LIN {X 0,Y 370.085,Z 646.724,A -85,B 0,C 180,E1 -12842.273,E2 -12842.273} C_VEL
LIN {X 0,Y 368.993,Z 653.125,A -85,B 0,C 180,E1 -12844.625,E2 -12844.625} C_VEL
LIN {X 0,Y 368.227,Z 658.236,A -85,B 0,C 180,E1 -12846.967,E2 -12846.967} C_VEL
LIN {X 0,Y 367.722,Z 662.415,A -85,B 0,C 180,E1 -12849.474,E2 -12849.474} C_VEL
LIN {X 0,Y 367.363,Z 665.468,A -85,B 0,C 180,E1 -12852.176,E2 -12852.176} C_VEL
LIN {X 0,Y 367.23,Z 666.86,A -85,B 0,C 180,E1 -12854.459,E2 -12854.459} C_VEL
LIN {X 0,Y 367.243,Z 667.317,A -85,B 0,C 180,E1 -12856.724,E2 -12856.724} C_VEL
LIN {X 0,Y 367.314,Z 666.714,A -85,B 0,C 180,E1 -12858.969,E2 -12858.969} C_VEL
LIN {X 0,Y 367.306,Z 665.194,A -85,B 0,C 180,E1 -12861.195,E2 -12861.195} C_VEL
LIN {X 0,Y 367.629,Z 662.16,A -85,B 0,C 180,E1 -12863.773,E2 -12863.773} C_VEL
LIN {X 0,Y 368.057,Z 656.967,A -85,B 0,C 180,E1 -12866.716,E2 -12866.716} C_VEL
LIN {X 0,Y 368.653,Z 650.369,A -85,B 0,C 180,E1 -12869.454,E2 -12869.454} C_VEL
LIN {X 0,Y 369.518,Z 643.703,A -85,B 0,C 180,E1 -12871.635,E2 -12871.635} C_VEL
LIN {X 0,Y 370.589,Z 635.761,A -85,B 0,C 180,E1 -12873.806,E2 -12873.806} C_VEL
LIN {X 0,Y 371.387,Z 631.353,A -85,B 0,C 180,E1 -12874.856,E2 -12874.856} C_VEL
LIN {X 0,Y 371.332,Z 628.098,A -85,B 0,C 180,E1 -12875.611,E2 -12875.611} C_VEL
LIN {X 0,Y 367.639,Z 616.959,A -85,B 0,C 180,E1 -12878.099,E2 -12878.099} C_VEL
LIN {X 0,Y 367.616,Z 613.116,A -85,B 0,C 180,E1 -12878.804,E2 -12878.804} C_VEL
LIN {X 0,Y 369.599,Z 601.168,A -85,B 0,C 180,E1 -12880.684,E2 -12880.684} C_VEL
LIN {X 0,Y 371.698,Z 588.051,A -85,B 0,C 180,E1 -12882.42,E2 -12882.42} C_VEL
LIN {X 0,Y 373.867,Z 573.601,A -85,B 0,C 180,E1 -12884.006,E2 -12884.006} C_VEL
LIN {X 0,Y 375.922,Z 559.065,A -85,B 0,C 180,E1 -12885.312,E2 -12885.312} C_VEL
LIN {X 0,Y 377.536,Z 545.128,A -85,B 0,C 180,E1 -12886.353,E2 -12886.353} C_VEL
LIN {X 0,Y 379.089,Z 530.243,A -85,B 0,C 180,E1 -12887.255,E2 -12887.255} C_VEL
LIN {X 0,Y 380.528,Z 513.702,A -85,B 0,C 180,E1 -12888.02,E2 -12888.02} C_VEL
LIN {X 0,Y 381.547,Z 498.273,A -85,B 0,C 180,E1 -12888.526,E2 -12888.526} C_VEL
LIN {X 0,Y 382.324,Z 475.986,A -85,B 0,C 180,E1 -12889.009,E2 -12889.009} C_VEL
LIN {X 0,Y 386.111,Z 337.639,A -85,B 0,C 180,E1 -12891.633,E2 -12891.633} C_VEL
LIN {X 0,Y 376.859,Z 317.995,A -85,B 0,C 180,E1 -12892.926,E2 -12892.926} C_VEL
LIN {X 0,Y 368.621,Z 302.126,A -85,B 0,C 180,E1 -12894.104,E2 -12894.104} C_VEL
LIN {X 0,Y 363.341,Z 293.257,A -85,B 0,C 180,E1 -12894.862,E2 -12894.862} C_VEL
LIN {X 0,Y 362.026,Z 290.544,A -85,B 0,C 180,E1 -12895.068,E2 -12895.068} C_VEL
LIN {X 0,Y 361.859,Z 289.711,A -85,B 0,C 180,E1 -12895.133,E2 -12895.133} C_VEL
LIN {X 0,Y 361.859,Z 289.723,A -85,B 0,C 180,E1 -12899.073,E2 -12899.073} C_VEL
LIN {X 0,Y 361.849,Z 289.725,A -85,B 0,C 180,E1 -12902.945,E2 -12902.945} C_VEL
LIN {X 0,Y 361.865,Z 289.716,A -85,B 0,C 180,E1 -12905.637,E2 -12905.637} C_VEL
LIN {X 0,Y 361.827,Z 289.722,A -85,B 0,C 180,E1 -12909.017,E2 -12909.017} C_VEL
LIN {X 0,Y 361.831,Z 289.72,A -85,B 0,C 180,E1 -12912.83,E2 -12912.83} C_VEL
LIN {X 0,Y 361.814,Z 289.718,A -85,B 0,C 180,E1 -12915.947,E2 -12915.947} C_VEL
LIN {X 0,Y 361.812,Z 289.728,A -85,B 0,C 180,E1 -12919.249,E2 -12919.249} C_VEL
LIN {X 0,Y 361.862,Z 289.676,A -85,B 0,C 180,E1 -12922.981,E2 -12922.981} C_VEL
LIN {X 0,Y 361.859,Z 289.717,A -85,B 0,C 180,E1 -12926.631,E2 -12926.631} C_VEL
LIN {X 0,Y 361.857,Z 289.715,A -85,B 0,C 180,E1 -12929.67,E2 -12929.67} C_VEL
LIN {X 0,Y 361.857,Z 289.724,A -85,B 0,C 180,E1 -12933.467,E2 -12933.467} C_VEL
LIN {X 0,Y 361.866,Z 289.709,A -85,B 0,C 180,E1 -12937.142,E2 -12937.142} C_VEL
LIN {X 0,Y 361.907,Z 289.711,A -85,B 0,C 180,E1 -12940.723,E2 -12940.723} C_VEL
LIN {X 0,Y 361.944,Z 289.711,A -85,B 0,C 180,E1 -12944.225,E2 -12944.225} C_VEL
LIN {X 0,Y 362,Z 289.699,A -85,B 0,C 180,E1 -12946.527,E2 -12946.527} C_VEL
LIN {X 0,Y 362.029,Z 289.7,A -85,B 0,C 180,E1 -12949.937,E2 -12949.937} C_VEL
LIN {X 0,Y 362.15,Z 289.675,A -85,B 0,C 180,E1 -12953.313,E2 -12953.313} C_VEL
LIN {X 0,Y 362.271,Z 289.67,A -85,B 0,C 180,E1 -12957.776,E2 -12957.776} C_VEL
LIN {X 0,Y 362.425,Z 289.634,A -85,B 0,C 180,E1 -12959.999,E2 -12959.999} C_VEL
LIN {X 0,Y 362.281,Z 289.667,A -85,B 0,C 180,E1 -12962.223,E2 -12962.223} C_VEL
LIN {X 0,Y 362.147,Z 289.665,A -85,B 0,C 180,E1 -12966.686,E2 -12966.686} C_VEL
LIN {X 0,Y 362.056,Z 289.688,A -85,B 0,C 180,E1 -12968.933,E2 -12968.933} C_VEL
LIN {X 0,Y 361.96,Z 289.704,A -85,B 0,C 180,E1 -12972.332,E2 -12972.332} C_VEL
LIN {X 0,Y 361.961,Z 289.71,A -85,B 0,C 180,E1 -12974.62,E2 -12974.62} C_VEL
LIN {X 0,Y 361.91,Z 289.715,A -85,B 0,C 180,E1 -12978.101,E2 -12978.101} C_VEL
LIN {X 0,Y 361.891,Z 289.717,A -85,B 0,C 180,E1 -12981.652,E2 -12981.652} C_VEL
LIN {X 0,Y 361.927,Z 289.714,A -85,B 0,C 180,E1 -12985.289,E2 -12985.289} C_VEL
LIN {X 0,Y 361.907,Z 289.713,A -85,B 0,C 180,E1 -12987.779,E2 -12987.779} C_VEL
LIN {X 0,Y 361.836,Z 289.727,A -85,B 0,C 180,E1 -12991.629,E2 -12991.629} C_VEL
LIN {X 0,Y 361.873,Z 289.716,A -85,B 0,C 180,E1 -12995.345,E2 -12995.345} C_VEL
LIN {X 0,Y 361.87,Z 289.724,A -85,B 0,C 180,E1 -12999.027,E2 -12999.027} C_VEL
LIN {X 0,Y 361.835,Z 289.73,A -85,B 0,C 180,E1 -13002.828,E2 -13002.828} C_VEL
LIN {X 0,Y 361.851,Z 289.726,A -85,B 0,C 180,E1 -13005.941,E2 -13005.941} C_VEL
LIN {X 0,Y 361.872,Z 289.883,A -85,B 0,C 180,E1 -13009.425,E2 -13009.425} C_VEL
LIN {X 0,Y 367.396,Z 306.317,A -85,B 0,C 180,E1 -13012.483,E2 -13012.483} C_VEL
LIN {X 0,Y 377.226,Z 326.254,A -85,B 0,C 180,E1 -13013.91,E2 -13013.91} C_VEL
LIN {X 0,Y 384.815,Z 343.06,A -85,B 0,C 180,E1 -13014.983,E2 -13014.983} C_VEL
LIN {X 0,Y 386.007,Z 350.145,A -85,B 0,C 180,E1 -13015.243,E2 -13015.243} C_VEL
LIN {X 0,Y 381.47,Z 514.209,A -85,B 0,C 180,E1 -13018.381,E2 -13018.381} C_VEL
LIN {X 0,Y 380.276,Z 531.49,A -85,B 0,C 180,E1 -13018.914,E2 -13018.914} C_VEL
LIN {X 0,Y 378.832,Z 547.72,A -85,B 0,C 180,E1 -13019.633,E2 -13019.633} C_VEL
LIN {X 0,Y 377.102,Z 563.635,A -85,B 0,C 180,E1 -13020.558,E2 -13020.558} C_VEL
LIN {X 0,Y 375.227,Z 578.232,A -85,B 0,C 180,E1 -13021.616,E2 -13021.616} C_VEL
LIN {X 0,Y 373.014,Z 593.418,A -85,B 0,C 180,E1 -13022.965,E2 -13022.965} C_VEL
LIN {X 0,Y 371.039,Z 607.253,A -85,B 0,C 180,E1 -13024.474,E2 -13024.474} C_VEL
LIN {X 0,Y 368.941,Z 619.349,A -85,B 0,C 180,E1 -13026.025,E2 -13026.025} C_VEL
LIN {X 0,Y 367.037,Z 630.986,A -85,B 0,C 180,E1 -13027.78,E2 -13027.78} C_VEL
LIN {X 0,Y 365.235,Z 642.007,A -85,B 0,C 180,E1 -13029.735,E2 -13029.735} C_VEL
LIN {X 0,Y 363.626,Z 652.593,A -85,B 0,C 180,E1 -13031.987,E2 -13031.987} C_VEL
LIN {X 0,Y 362.341,Z 661.434,A -85,B 0,C 180,E1 -13034.244,E2 -13034.244} C_VEL
LIN {X 0,Y 361.504,Z 668.814,A -85,B 0,C 180,E1 -13036.509,E2 -13036.509} C_VEL
LIN {X 0,Y 360.867,Z 674.908,A -85,B 0,C 180,E1 -13038.77,E2 -13038.77} C_VEL
LIN {X 0,Y 360.456,Z 680.797,A -85,B 0,C 180,E1 -13041.592,E2 -13041.592} C_VEL
LIN {X 0,Y 360.374,Z 684.478,A -85,B 0,C 180,E1 -13044.038,E2 -13044.038} C_VEL
LIN {X 0,Y 360.28,Z 687.094,A -85,B 0,C 180,E1 -13046.645,E2 -13046.645} C_VEL
LIN {X 0,Y 360.315,Z 688.304,A -85,B 0,C 180,E1 -13048.882,E2 -13048.882} C_VEL
LIN {X 0,Y 360.315,Z 688.465,A -85,B 0,C 180,E1 -13051.118,E2 -13051.118} C_VEL
LIN {X 0,Y 360.274,Z 687.726,A -85,B 0,C 180,E1 -13053.355,E2 -13053.355} C_VEL
LIN {X 0,Y 360.374,Z 685.579,A -85,B 0,C 180,E1 -13055.962,E2 -13055.962} C_VEL
LIN {X 0,Y 360.45,Z 683.261,A -85,B 0,C 180,E1 -13057.845,E2 -13057.845} C_VEL
LIN {X 0,Y 360.666,Z 679.474,A -85,B 0,C 180,E1 -13060.101,E2 -13060.101} C_VEL
LIN {X 0,Y 361.249,Z 674.706,A -85,B 0,C 180,E1 -13062.357,E2 -13062.357} C_VEL
LIN {X 0,Y 362.007,Z 668.696,A -85,B 0,C 180,E1 -13064.619,E2 -13064.619} C_VEL
LIN {X 0,Y 363.453,Z 660.481,A -85,B 0,C 180,E1 -13067.151,E2 -13067.151} C_VEL
LIN {X 0,Y 365.086,Z 651.689,A -85,B 0,C 180,E1 -13069.395,E2 -13069.395} C_VEL
LIN {X 0,Y 367.174,Z 641.258,A -85,B 0,C 180,E1 -13071.621,E2 -13071.621} C_VEL
LIN {X 0,Y 369.626,Z 629.387,A -85,B 0,C 180,E1 -13073.732,E2 -13073.732} C_VEL
LIN {X 0,Y 371.938,Z 617.815,A -85,B 0,C 180,E1 -13075.46,E2 -13075.46} C_VEL
LIN {X 0,Y 374.42,Z 605.077,A -85,B 0,C 180,E1 -13077.077,E2 -13077.077} C_VEL
LIN {X 0,Y 377.087,Z 591.395,A -85,B 0,C 180,E1 -13078.523,E2 -13078.523} C_VEL
LIN {X 0,Y 379.398,Z 578,A -85,B 0,C 180,E1 -13079.704,E2 -13079.704} C_VEL
LIN {X 0,Y 381.636,Z 563.787,A -85,B 0,C 180,E1 -13080.733,E2 -13080.733} C_VEL
LIN {X 0,Y 383.646,Z 548.604,A -85,B 0,C 180,E1 -13081.627,E2 -13081.627} C_VEL
LIN {X 0,Y 385.281,Z 533.349,A -85,B 0,C 180,E1 -13082.323,E2 -13082.323} C_VEL
LIN {X 0,Y 386.645,Z 517.043,A -85,B 0,C 180,E1 -13082.852,E2 -13082.852} C_VEL
LIN {X 0,Y 387.657,Z 494.521,A -85,B 0,C 180,E1 -13083.334,E2 -13083.334} C_VEL
LIN {X 0,Y 392.435,Z 351.432,A -85,B 0,C 180,E1 -13086.098,E2 -13086.098} C_VEL
LIN {X 0,Y 391.864,Z 348.162,A -85,B 0,C 180,E1 -13086.244,E2 -13086.244} C_VEL
LIN {X 0,Y 383.625,Z 331.703,A -85,B 0,C 180,E1 -13087.688,E2 -13087.688} C_VEL
LIN {X 0,Y 374.037,Z 314.955,A -85,B 0,C 180,E1 -13089.44,E2 -13089.44} C_VEL
LIN {X 0,Y 367.91,Z 304.9,A -85,B 0,C 180,E1 -13090.637,E2 -13090.637} C_VEL
LIN {X 0,Y 363.24,Z 293.204,A -85,B 0,C 180,E1 -13093.486,E2 -13093.486} C_VEL
LIN {X 0,Y 362.102,Z 290.962,A -85,B 0,C 180,E1 -13094.1,E2 -13094.1} C_VEL
LIN {X 0,Y 361.829,Z 289.716,A -85,B 0,C 180,E1 -13094.409,E2 -13094.409} C_VEL
LIN {X 0,Y 361.835,Z 289.718,A -85,B 0,C 180,E1 -13097.569,E2 -13097.569} C_VEL
LIN {X 0,Y 361.87,Z 289.72,A -85,B 0,C 180,E1 -13100.974,E2 -13100.974} C_VEL
LIN {X 0,Y 361.874,Z 289.722,A -85,B 0,C 180,E1 -13104.656,E2 -13104.656} C_VEL
LIN {X 0,Y 361.837,Z 289.718,A -85,B 0,C 180,E1 -13108.371,E2 -13108.371} C_VEL
LIN {X 0,Y 361.908,Z 289.691,A -85,B 0,C 180,E1 -13112.222,E2 -13112.222} C_VEL
LIN {X 0,Y 361.928,Z 289.716,A -85,B 0,C 180,E1 -13114.711,E2 -13114.711} C_VEL
LIN {X 0,Y 361.862,Z 289.702,A -85,B 0,C 180,E1 -13118.346,E2 -13118.346} C_VEL
LIN {X 0,Y 361.968,Z 289.689,A -85,B 0,C 180,E1 -13122.062,E2 -13122.062} C_VEL
LIN {X 0,Y 361.999,Z 289.705,A -85,B 0,C 180,E1 -13126.102,E2 -13126.102} C_VEL
LIN {X 0,Y 362.001,Z 289.676,A -85,B 0,C 180,E1 -13129.938,E2 -13129.938} C_VEL
LIN {X 0,Y 362.126,Z 289.686,A -85,B 0,C 180,E1 -13133.314,E2 -13133.314} C_VEL
LIN {X 0,Y 362.274,Z 289.665,A -85,B 0,C 180,E1 -13137.777,E2 -13137.777} C_VEL
LIN {X 0,Y 362.363,Z 289.652,A -85,B 0,C 180,E1 -13140.001,E2 -13140.001} C_VEL
LIN {X 0,Y 362.267,Z 289.642,A -85,B 0,C 180,E1 -13142.224,E2 -13142.224} C_VEL
LIN {X 0,Y 362.126,Z 289.675,A -85,B 0,C 180,E1 -13146.688,E2 -13146.688} C_VEL
LIN {X 0,Y 362.002,Z 289.698,A -85,B 0,C 180,E1 -13150.063,E2 -13150.063} C_VEL
LIN {X 0,Y 361.998,Z 289.68,A -85,B 0,C 180,E1 -13153.897,E2 -13153.897} C_VEL
LIN {X 0,Y 361.907,Z 289.703,A -85,B 0,C 180,E1 -13157.908,E2 -13157.908} C_VEL
LIN {X 0,Y 361.856,Z 289.724,A -85,B 0,C 180,E1 -13161.656,E2 -13161.656} C_VEL
LIN {X 0,Y 361.853,Z 289.717,A -85,B 0,C 180,E1 -13165.296,E2 -13165.296} C_VEL
LIN {X 0,Y 361.858,Z 289.711,A -85,B 0,C 180,E1 -13169.074,E2 -13169.074} C_VEL
LIN {X 0,Y 361.848,Z 289.716,A -85,B 0,C 180,E1 -13172.946,E2 -13172.946} C_VEL
LIN {X 0,Y 361.892,Z 289.833,A -85,B 0,C 180,E1 -13175.384,E2 -13175.384} C_VEL
LIN {X 0,Y 362.168,Z 291.049,A -85,B 0,C 180,E1 -13175.523,E2 -13175.523} C_VEL
LIN {X 0,Y 363.591,Z 293.551,A -85,B 0,C 180,E1 -13175.826,E2 -13175.826} C_VEL
LIN {X 0,Y 365.132,Z 295.168,A -85,B 0,C 180,E1 -13176.12,E2 -13176.12} C_VEL
LIN {X 0,Y 367.269,Z 298.449,A -85,B 0,C 180,E1 -13176.547,E2 -13176.547} C_VEL
LIN {X 0,Y 368.815,Z 300.614,A -85,B 0,C 180,E1 -13176.845,E2 -13176.845} C_VEL
LIN {X 0,Y 375.341,Z 310.469,A -85,B 0,C 180,E1 -13178.079,E2 -13178.079} C_VEL
LIN {X 0,Y 384.501,Z 325.897,A -85,B 0,C 180,E1 -13179.732,E2 -13179.732} C_VEL
LIN {X 0,Y 392.18,Z 340.4,A -85,B 0,C 180,E1 -13181.059,E2 -13181.059} C_VEL
LIN {X 0,Y 392.754,Z 342.072,A -85,B 0,C 180,E1 -13181.168,E2 -13181.168} C_VEL
LIN {X 0,Y 387.371,Z 494.991,A -85,B 0,C 180,E1 -13184.129,E2 -13184.129} C_VEL
LIN {X 0,Y 386.172,Z 511.607,A -85,B 0,C 180,E1 -13184.645,E2 -13184.645} C_VEL
LIN {X 0,Y 384.687,Z 527.207,A -85,B 0,C 180,E1 -13185.332,E2 -13185.332} C_VEL
LIN {X 0,Y 382.808,Z 542.708,A -85,B 0,C 180,E1 -13186.219,E2 -13186.219} C_VEL
LIN {X 0,Y 380.595,Z 558.256,A -85,B 0,C 180,E1 -13187.344,E2 -13187.344} C_VEL
LIN {X 0,Y 378.051,Z 573.475,A -85,B 0,C 180,E1 -13188.704,E2 -13188.704} C_VEL
LIN {X 0,Y 375.458,Z 587.611,A -85,B 0,C 180,E1 -13190.255,E2 -13190.255} C_VEL
LIN {X 0,Y 372.987,Z 599.87,A -85,B 0,C 180,E1 -13191.859,E2 -13191.859} C_VEL
LIN {X 0,Y 370.544,Z 611.483,A -85,B 0,C 180,E1 -13193.65,E2 -13193.65} C_VEL
LIN {X 0,Y 368.1,Z 622.784,A -85,B 0,C 180,E1 -13195.72,E2 -13195.72} C_VEL
LIN {X 0,Y 366.207,Z 631.926,A -85,B 0,C 180,E1 -13197.723,E2 -13197.723} C_VEL
LIN {X 0,Y 364.464,Z 640.359,A -85,B 0,C 180,E1 -13199.91,E2 -13199.91} C_VEL
LIN {X 0,Y 363.019,Z 648.046,A -85,B 0,C 180,E1 -13202.313,E2 -13202.313} C_VEL
LIN {X 0,Y 361.908,Z 654.301,A -85,B 0,C 180,E1 -13204.708,E2 -13204.708} C_VEL
LIN {X 0,Y 361.128,Z 659.165,A -85,B 0,C 180,E1 -13207.094,E2 -13207.094} C_VEL
LIN {X 0,Y 360.662,Z 662.879,A -85,B 0,C 180,E1 -13209.466,E2 -13209.466} C_VEL
LIN {X 0,Y 360.294,Z 665.481,A -85,B 0,C 180,E1 -13211.814,E2 -13211.814} C_VEL
LIN {X 0,Y 360.166,Z 666.985,A -85,B 0,C 180,E1 -13214.146,E2 -13214.146} C_VEL
LIN {X 0,Y 360.141,Z 667.536,A -85,B 0,C 180,E1 -13216.457,E2 -13216.457} C_VEL
LIN {X 0,Y 360.213,Z 667.008,A -85,B 0,C 180,E1 -13218.749,E2 -13218.749} C_VEL
LIN {X 0,Y 360.193,Z 665.597,A -85,B 0,C 180,E1 -13221.02,E2 -13221.02} C_VEL
LIN {X 0,Y 360.548,Z 662.44,A -85,B 0,C 180,E1 -13223.79,E2 -13223.79} C_VEL
LIN {X 0,Y 360.785,Z 658.621,A -85,B 0,C 180,E1 -13226.09,E2 -13226.09} C_VEL
LIN {X 0,Y 361.245,Z 653.894,A -85,B 0,C 180,E1 -13228.328,E2 -13228.328} C_VEL
LIN {X 0,Y 362.035,Z 647.944,A -85,B 0,C 180,E1 -13230.556,E2 -13230.556} C_VEL
LIN {X 0,Y 362.947,Z 640.796,A -85,B 0,C 180,E1 -13232.775,E2 -13232.775} C_VEL
LIN {X 0,Y 364.431,Z 631.914,A -85,B 0,C 180,E1 -13235.058,E2 -13235.058} C_VEL
LIN {X 0,Y 366.144,Z 622.083,A -85,B 0,C 180,E1 -13237.167,E2 -13237.167} C_VEL
LIN {X 0,Y 367.616,Z 613.116,A -85,B 0,C 180,E1 -13238.804,E2 -13238.804} C_VEL
LIN {X 0,Y 367.632,Z 609.268,A -85,B 0,C 180,E1 -13239.492,E2 -13239.492} C_VEL
LIN {X 0,Y 364.64,Z 597.528,A -85,B 0,C 180,E1 -13241.553,E2 -13241.553} C_VEL
LIN {X 0,Y 364.371,Z 593.241,A -85,B 0,C 180,E1 -13242.193,E2 -13242.193} C_VEL
LIN {X 0,Y 364.532,Z 591.722,A -85,B 0,C 180,E1 -13242.394,E2 -13242.394} C_VEL
LIN {X 0,Y 366.676,Z 578.023,A -85,B 0,C 180,E1 -13244.003,E2 -13244.003} C_VEL
LIN {X 0,Y 368.775,Z 564.409,A -85,B 0,C 180,E1 -13245.333,E2 -13245.333} C_VEL
LIN {X 0,Y 370.719,Z 549.691,A -85,B 0,C 180,E1 -13246.521,E2 -13246.521} C_VEL
LIN {X 0,Y 372.287,Z 534.616,A -85,B 0,C 180,E1 -13247.51,E2 -13247.51} C_VEL
LIN {X 0,Y 373.878,Z 518.564,A -85,B 0,C 180,E1 -13248.317,E2 -13248.317} C_VEL
LIN {X 0,Y 374.962,Z 503.284,A -85,B 0,C 180,E1 -13248.899,E2 -13248.899} C_VEL
LIN {X 0,Y 375.802,Z 486.805,A -85,B 0,C 180,E1 -13249.316,E2 -13249.316} C_VEL
LIN {X 0,Y 380.045,Z 340.707,A -85,B 0,C 180,E1 -13252.121,E2 -13252.121} C_VEL
LIN {X 0,Y 379.559,Z 338.843,A -85,B 0,C 180,E1 -13252.207,E2 -13252.207} C_VEL
LIN {X 0,Y 370.999,Z 320.605,A -85,B 0,C 180,E1 -13253.441,E2 -13253.441} C_VEL
LIN {X 0,Y 362.905,Z 305.09,A -85,B 0,C 180,E1 -13254.63,E2 -13254.63} C_VEL
LIN {X 0,Y 356.402,Z 294.254,A -85,B 0,C 180,E1 -13255.597,E2 -13255.597} C_VEL
LIN {X 0,Y 355.008,Z 291.577,A -85,B 0,C 180,E1 -13255.819,E2 -13255.819} C_VEL
LIN {X 0,Y 354.823,Z 290.582,A -85,B 0,C 180,E1 -13255.903,E2 -13255.903} C_VEL
LIN {X 0,Y 354.796,Z 290.602,A -85,B 0,C 180,E1 -13259.684,E2 -13259.684} C_VEL
LIN {X 0,Y 354.81,Z 290.604,A -85,B 0,C 180,E1 -13263.702,E2 -13263.702} C_VEL
LIN {X 0,Y 354.795,Z 290.604,A -85,B 0,C 180,E1 -13266.46,E2 -13266.46} C_VEL
LIN {X 0,Y 354.771,Z 290.602,A -85,B 0,C 180,E1 -13269.412,E2 -13269.412} C_VEL
LIN {X 0,Y 354.783,Z 290.598,A -85,B 0,C 180,E1 -13272.865,E2 -13272.865} C_VEL
LIN {X 0,Y 354.763,Z 290.595,A -85,B 0,C 180,E1 -13276.102,E2 -13276.102} C_VEL
LIN {X 0,Y 354.764,Z 290.606,A -85,B 0,C 180,E1 -13279.175,E2 -13279.175} C_VEL
LIN {X 0,Y 354.8,Z 290.56,A -85,B 0,C 180,E1 -13282.404,E2 -13282.404} C_VEL
LIN {X 0,Y 354.809,Z 290.568,A -85,B 0,C 180,E1 -13284.94,E2 -13284.94} C_VEL
LIN {X 0,Y 354.795,Z 290.601,A -85,B 0,C 180,E1 -13288.405,E2 -13288.405} C_VEL
LIN {X 0,Y 354.798,Z 290.59,A -85,B 0,C 180,E1 -13291.614,E2 -13291.614} C_VEL
LIN {X 0,Y 354.835,Z 290.585,A -85,B 0,C 180,E1 -13295.657,E2 -13295.657} C_VEL
LIN {X 0,Y 354.828,Z 290.598,A -85,B 0,C 180,E1 -13299.113,E2 -13299.113} C_VEL
LIN {X 0,Y 354.881,Z 290.578,A -85,B 0,C 180,E1 -13302.718,E2 -13302.718} C_VEL
LIN {X 0,Y 354.953,Z 290.578,A -85,B 0,C 180,E1 -13306.255,E2 -13306.255} C_VEL
LIN {X 0,Y 354.977,Z 290.574,A -85,B 0,C 180,E1 -13309.735,E2 -13309.735} C_VEL
LIN {X 0,Y 355.113,Z 290.553,A -85,B 0,C 180,E1 -13313.18,E2 -13313.18} C_VEL
LIN {X 0,Y 355.234,Z 290.547,A -85,B 0,C 180,E1 -13317.732,E2 -13317.732} C_VEL
LIN {X 0,Y 355.374,Z 290.512,A -85,B 0,C 180,E1 -13319.999,E2 -13319.999} C_VEL
LIN {X 0,Y 355.244,Z 290.543,A -85,B 0,C 180,E1 -13322.267,E2 -13322.267} C_VEL
LIN {X 0,Y 355.113,Z 290.54,A -85,B 0,C 180,E1 -13326.819,E2 -13326.819} C_VEL
LIN {X 0,Y 355.004,Z 290.568,A -85,B 0,C 180,E1 -13329.112,E2 -13329.112} C_VEL
LIN {X 0,Y 354.921,Z 290.581,A -85,B 0,C 180,E1 -13332.58,E2 -13332.58} C_VEL
LIN {X 0,Y 354.886,Z 290.588,A -85,B 0,C 180,E1 -13336.096,E2 -13336.096} C_VEL
LIN {X 0,Y 354.856,Z 290.596,A -85,B 0,C 180,E1 -13339.675,E2 -13339.675} C_VEL
LIN {X 0,Y 354.832,Z 290.602,A -85,B 0,C 180,E1 -13343.336,E2 -13343.336} C_VEL
LIN {X 0,Y 354.886,Z 290.596,A -85,B 0,C 180,E1 -13346.981,E2 -13346.981} C_VEL
LIN {X 0,Y 354.816,Z 290.601,A -85,B 0,C 180,E1 -13349.681,E2 -13349.681} C_VEL
LIN {X 0,Y 354.804,Z 290.601,A -85,B 0,C 180,E1 -13353.702,E2 -13353.702} C_VEL
LIN {X 0,Y 354.797,Z 290.59,A -85,B 0,C 180,E1 -13356.459,E2 -13356.459} C_VEL
LIN {X 0,Y 354.822,Z 290.598,A -85,B 0,C 180,E1 -13359.423,E2 -13359.423} C_VEL
LIN {X 0,Y 354.786,Z 290.607,A -85,B 0,C 180,E1 -13362.867,E2 -13362.867} C_VEL
LIN {X 0,Y 354.794,Z 290.606,A -85,B 0,C 180,E1 -13366.108,E2 -13366.108} C_VEL
LIN {X 0,Y 354.808,Z 290.75,A -85,B 0,C 180,E1 -13368.754,E2 -13368.754} C_VEL
LIN {X 0,Y 359.949,Z 305.875,A -85,B 0,C 180,E1 -13371.688,E2 -13371.688} C_VEL
LIN {X 0,Y 370.514,Z 327.049,A -85,B 0,C 180,E1 -13373.275,E2 -13373.275} C_VEL
LIN {X 0,Y 379.013,Z 345.632,A -85,B 0,C 180,E1 -13374.508,E2 -13374.508} C_VEL
LIN {X 0,Y 379.921,Z 351.835,A -85,B 0,C 180,E1 -13374.728,E2 -13374.728} C_VEL
LIN {X 0,Y 375.254,Z 513.016,A -85,B 0,C 180,E1 -13377.849,E2 -13377.849} C_VEL
LIN {X 0,Y 374.154,Z 529.424,A -85,B 0,C 180,E1 -13378.347,E2 -13378.347} C_VEL
LIN {X 0,Y 372.761,Z 544.864,A -85,B 0,C 180,E1 -13379.006,E2 -13379.006} C_VEL
LIN {X 0,Y 371.128,Z 560.404,A -85,B 0,C 180,E1 -13379.879,E2 -13379.879} C_VEL
LIN {X 0,Y 369.126,Z 575.609,A -85,B 0,C 180,E1 -13380.955,E2 -13380.955} C_VEL
LIN {X 0,Y 366.897,Z 591.109,A -85,B 0,C 180,E1 -13382.321,E2 -13382.321} C_VEL
LIN {X 0,Y 364.804,Z 604.075,A -85,B 0,C 180,E1 -13383.698,E2 -13383.698} C_VEL
LIN {X 0,Y 362.691,Z 616.641,A -85,B 0,C 180,E1 -13385.272,E2 -13385.272} C_VEL
LIN {X 0,Y 360.684,Z 628.685,A -85,B 0,C 180,E1 -13387.064,E2 -13387.064} C_VEL
LIN {X 0,Y 358.691,Z 639.94,A -85,B 0,C 180,E1 -13389.048,E2 -13389.048} C_VEL
LIN {X 0,Y 357.087,Z 650.106,A -85,B 0,C 180,E1 -13391.174,E2 -13391.174} C_VEL
LIN {X 0,Y 355.697,Z 658.932,A -85,B 0,C 180,E1 -13393.352,E2 -13393.352} C_VEL
LIN {X 0,Y 354.698,Z 666.72,A -85,B 0,C 180,E1 -13395.66,E2 -13395.66} C_VEL
LIN {X 0,Y 353.978,Z 673.096,A -85,B 0,C 180,E1 -13397.967,E2 -13397.967} C_VEL
LIN {X 0,Y 353.486,Z 678.302,A -85,B 0,C 180,E1 -13400.271,E2 -13400.271} C_VEL
LIN {X 0,Y 353.356,Z 681.419,A -85,B 0,C 180,E1 -13401.997,E2 -13401.997} C_VEL
LIN {X 0,Y 353.258,Z 684.674,A -85,B 0,C 180,E1 -13404.291,E2 -13404.291} C_VEL
LIN {X 0,Y 353.201,Z 686.845,A -85,B 0,C 180,E1 -13406.578,E2 -13406.578} C_VEL
LIN {X 0,Y 353.216,Z 688.071,A -85,B 0,C 180,E1 -13408.86,E2 -13408.86} C_VEL
LIN {X 0,Y 353.214,Z 688.265,A -85,B 0,C 180,E1 -13411.14,E2 -13411.14} C_VEL
LIN {X 0,Y 353.194,Z 687.543,A -85,B 0,C 180,E1 -13413.422,E2 -13413.422} C_VEL
LIN {X 0,Y 353.273,Z 685.605,A -85,B 0,C 180,E1 -13415.908,E2 -13415.908} C_VEL
LIN {X 0,Y 353.361,Z 683.132,A -85,B 0,C 180,E1 -13418.003,E2 -13418.003} C_VEL
LIN {X 0,Y 353.754,Z 678.308,A -85,B 0,C 180,E1 -13420.879,E2 -13420.879} C_VEL
LIN {X 0,Y 354.465,Z 673.229,A -85,B 0,C 180,E1 -13423.18,E2 -13423.18} C_VEL
LIN {X 0,Y 355.368,Z 667.045,A -85,B 0,C 180,E1 -13425.485,E2 -13425.485} C_VEL
LIN {X 0,Y 357.041,Z 658.483,A -85,B 0,C 180,E1 -13428.061,E2 -13428.061} C_VEL
LIN {X 0,Y 358.791,Z 649.315,A -85,B 0,C 180,E1 -13430.346,E2 -13430.346} C_VEL
LIN {X 0,Y 361.153,Z 638.455,A -85,B 0,C 180,E1 -13432.602,E2 -13432.602} C_VEL
LIN {X 0,Y 363.594,Z 627.204,A -85,B 0,C 180,E1 -13434.569,E2 -13434.569} C_VEL
LIN {X 0,Y 366.182,Z 615.169,A -85,B 0,C 180,E1 -13436.349,E2 -13436.349} C_VEL
LIN {X 0,Y 368.615,Z 603.11,A -85,B 0,C 180,E1 -13437.847,E2 -13437.847} C_VEL
LIN {X 0,Y 371.353,Z 589.187,A -85,B 0,C 180,E1 -13439.303,E2 -13439.303} C_VEL
LIN {X 0,Y 373.815,Z 575.398,A -85,B 0,C 180,E1 -13440.506,E2 -13440.506} C_VEL
LIN {X 0,Y 376.481,Z 558.69,A -85,B 0,C 180,E1 -13441.67,E2 -13441.67} C_VEL
LIN {X 0,Y 378.565,Z 542.077,A -85,B 0,C 180,E1 -13442.574,E2 -13442.574} C_VEL
LIN {X 0,Y 380.194,Z 527.12,A -85,B 0,C 180,E1 -13443.165,E2 -13443.165} C_VEL
LIN {X 0,Y 381.309,Z 512.461,A -85,B 0,C 180,E1 -13443.598,E2 -13443.598} C_VEL
LIN {X 0,Y 386.963,Z 353.291,A -85,B 0,C 180,E1 -13446.73,E2 -13446.73} C_VEL
LIN {X 0,Y 386.544,Z 351.056,A -85,B 0,C 180,E1 -13446.837,E2 -13446.837} C_VEL
LIN {X 0,Y 379.203,Z 336.245,A -85,B 0,C 180,E1 -13448.168,E2 -13448.168} C_VEL
LIN {X 0,Y 369.989,Z 319.961,A -85,B 0,C 180,E1 -13449.904,E2 -13449.904} C_VEL
LIN {X 0,Y 362.878,Z 308.558,A -85,B 0,C 180,E1 -13451.316,E2 -13451.316} C_VEL
LIN {X 0,Y 360.362,Z 304.462,A -85,B 0,C 180,E1 -13451.873,E2 -13451.873} C_VEL
LIN {X 0,Y 355.877,Z 293.535,A -85,B 0,C 180,E1 -13454.689,E2 -13454.689} C_VEL
LIN {X 0,Y 354.791,Z 290.59,A -85,B 0,C 180,E1 -13455.489,E2 -13455.489} C_VEL
LIN {X 0,Y 354.786,Z 290.589,A -85,B 0,C 180,E1 -13459.18,E2 -13459.18} C_VEL
LIN {X 0,Y 354.807,Z 290.583,A -85,B 0,C 180,E1 -13462.403,E2 -13462.403} C_VEL
LIN {X 0,Y 354.812,Z 290.601,A -85,B 0,C 180,E1 -13464.941,E2 -13464.941} C_VEL
LIN {X 0,Y 354.793,Z 290.595,A -85,B 0,C 180,E1 -13468.406,E2 -13468.406} C_VEL
LIN {X 0,Y 354.846,Z 290.57,A -85,B 0,C 180,E1 -13471.619,E2 -13471.619} C_VEL
LIN {X 0,Y 354.899,Z 290.588,A -85,B 0,C 180,E1 -13474.173,E2 -13474.173} C_VEL
LIN {X 0,Y 354.817,Z 290.574,A -85,B 0,C 180,E1 -13477.893,E2 -13477.893} C_VEL
LIN {X 0,Y 354.924,Z 290.569,A -85,B 0,C 180,E1 -13481.892,E2 -13481.892} C_VEL
LIN {X 0,Y 354.944,Z 290.583,A -85,B 0,C 180,E1 -13485.982,E2 -13485.982} C_VEL
LIN {X 0,Y 354.957,Z 290.551,A -85,B 0,C 180,E1 -13489.736,E2 -13489.736} C_VEL
LIN {X 0,Y 355.091,Z 290.563,A -85,B 0,C 180,E1 -13493.18,E2 -13493.18} C_VEL
LIN {X 0,Y 355.236,Z 290.542,A -85,B 0,C 180,E1 -13497.733,E2 -13497.733} C_VEL
LIN {X 0,Y 355.315,Z 290.529,A -85,B 0,C 180,E1 -13500.001,E2 -13500.001} C_VEL
LIN {X 0,Y 355.229,Z 290.518,A -85,B 0,C 180,E1 -13502.268,E2 -13502.268} C_VEL
LIN {X 0,Y 355.091,Z 290.548,A -85,B 0,C 180,E1 -13506.821,E2 -13506.821} C_VEL
LIN {X 0,Y 354.958,Z 290.578,A -85,B 0,C 180,E1 -13510.265,E2 -13510.265} C_VEL
LIN {X 0,Y 354.94,Z 290.558,A -85,B 0,C 180,E1 -13514.016,E2 -13514.016} C_VEL
LIN {X 0,Y 354.847,Z 290.579,A -85,B 0,C 180,E1 -13518.07,E2 -13518.07} C_VEL
LIN {X 0,Y 354.808,Z 290.599,A -85,B 0,C 180,E1 -13522.108,E2 -13522.108} C_VEL
LIN {X 0,Y 354.797,Z 290.602,A -85,B 0,C 180,E1 -13525.836,E2 -13525.836} C_VEL
LIN {X 0,Y 354.795,Z 290.599,A -85,B 0,C 180,E1 -13529.685,E2 -13529.685} C_VEL
LIN {X 0,Y 354.81,Z 290.604,A -85,B 0,C 180,E1 -13533.702,E2 -13533.702} C_VEL
LIN {X 0,Y 354.806,Z 290.602,A -85,B 0,C 180,E1 -13534.241,E2 -13534.241} C_VEL
LIN {X 0,Y 355.81,Z 293.459,A -85,B 0,C 180,E1 -13534.517,E2 -13534.517} C_VEL
LIN {X 0,Y 357.908,Z 295.591,A -85,B 0,C 180,E1 -13534.94,E2 -13534.94} C_VEL
LIN {X 0,Y 360.241,Z 299.311,A -85,B 0,C 180,E1 -13535.439,E2 -13535.439} C_VEL
LIN {X 0,Y 361.6,Z 300.988,A -85,B 0,C 180,E1 -13535.711,E2 -13535.711} C_VEL
LIN {X 0,Y 368.679,Z 311.327,A -85,B 0,C 180,E1 -13537.114,E2 -13537.114} C_VEL
LIN {X 0,Y 377.434,Z 325.766,A -85,B 0,C 180,E1 -13538.77,E2 -13538.77} C_VEL
LIN {X 0,Y 385.685,Z 340.953,A -85,B 0,C 180,E1 -13540.255,E2 -13540.255} C_VEL
LIN {X 0,Y 387.248,Z 344.132,A -85,B 0,C 180,E1 -13540.532,E2 -13540.532} C_VEL
LIN {X 0,Y 381.686,Z 495.648,A -85,B 0,C 180,E1 -13543.504,E2 -13543.504} C_VEL
LIN {X 0,Y 380.49,Z 511.658,A -85,B 0,C 180,E1 -13544.01,E2 -13544.01} C_VEL
LIN {X 0,Y 378.898,Z 527.509,A -85,B 0,C 180,E1 -13544.712,E2 -13544.712} C_VEL
LIN {X 0,Y 376.898,Z 543.343,A -85,B 0,C 180,E1 -13545.632,E2 -13545.632} C_VEL
LIN {X 0,Y 374.601,Z 558.783,A -85,B 0,C 180,E1 -13546.769,E2 -13546.769} C_VEL
LIN {X 0,Y 372.103,Z 573.209,A -85,B 0,C 180,E1 -13548.076,E2 -13548.076} C_VEL
LIN {X 0,Y 369.522,Z 586.482,A -85,B 0,C 180,E1 -13549.533,E2 -13549.533} C_VEL
LIN {X 0,Y 366.72,Z 599.948,A -85,B 0,C 180,E1 -13551.3,E2 -13551.3} C_VEL
LIN {X 0,Y 364.009,Z 612.259,A -85,B 0,C 180,E1 -13553.236,E2 -13553.236} C_VEL
LIN {X 0,Y 361.451,Z 623.491,A -85,B 0,C 180,E1 -13555.345,E2 -13555.345} C_VEL
LIN {X 0,Y 359.256,Z 633.577,A -85,B 0,C 180,E1 -13557.622,E2 -13557.622} C_VEL
LIN {X 0,Y 357.401,Z 641.974,A -85,B 0,C 180,E1 -13559.91,E2 -13559.91} C_VEL
LIN {X 0,Y 355.936,Z 649.254,A -85,B 0,C 180,E1 -13562.314,E2 -13562.314} C_VEL
LIN {X 0,Y 354.794,Z 655.364,A -85,B 0,C 180,E1 -13564.793,E2 -13564.793} C_VEL
LIN {X 0,Y 354.028,Z 660.098,A -85,B 0,C 180,E1 -13567.225,E2 -13567.225} C_VEL
LIN {X 0,Y 353.617,Z 662.893,A -85,B 0,C 180,E1 -13569.086,E2 -13569.086} C_VEL
LIN {X 0,Y 353.246,Z 665.495,A -85,B 0,C 180,E1 -13571.438,E2 -13571.438} C_VEL
LIN {X 0,Y 353.102,Z 667.112,A -85,B 0,C 180,E1 -13573.82,E2 -13573.82} C_VEL
LIN {X 0,Y 353.037,Z 667.719,A -85,B 0,C 180,E1 -13576.179,E2 -13576.179} C_VEL
LIN {X 0,Y 353.11,Z 667.3,A -85,B 0,C 180,E1 -13578.52,E2 -13578.52} C_VEL
LIN {X 0,Y 353.096,Z 665.953,A -85,B 0,C 180,E1 -13580.838,E2 -13580.838} C_VEL
LIN {X 0,Y 353.456,Z 662.695,A -85,B 0,C 180,E1 -13583.824,E2 -13583.824} C_VEL
LIN {X 0,Y 353.677,Z 659.191,A -85,B 0,C 180,E1 -13586.012,E2 -13586.012} C_VEL
LIN {X 0,Y 354.165,Z 654.548,A -85,B 0,C 180,E1 -13588.294,E2 -13588.294} C_VEL
LIN {X 0,Y 355.207,Z 647.098,A -85,B 0,C 180,E1 -13591.134,E2 -13591.134} C_VEL
LIN {X 0,Y 356.359,Z 638.7,A -85,B 0,C 180,E1 -13593.675,E2 -13593.675} C_VEL
LIN {X 0,Y 357.985,Z 629.655,A -85,B 0,C 180,E1 -13595.916,E2 -13595.916} C_VEL
LIN {X 0,Y 359.915,Z 618.94,A -85,B 0,C 180,E1 -13598.139,E2 -13598.139} C_VEL
LIN {X 0,Y 361.792,Z 607.93,A -85,B 0,C 180,E1 -13600.069,E2 -13600.069} C_VEL
LIN {X 0,Y 363.701,Z 596.924,A -85,B 0,C 180,E1 -13601.706,E2 -13601.706} C_VEL
LIN {X 0,Y 364.532,Z 591.722,A -85,B 0,C 180,E1 -13602.394,E2 -13602.394} C_VEL
LIN {X 0,Y 364.628,Z 587.278,A -85,B 0,C 180,E1 -13602.999,E2 -13602.999} C_VEL
LIN {X 0,Y 361.735,Z 572.447,A -85,B 0,C 180,E1 -13605.012,E2 -13605.012} C_VEL
LIN {X 0,Y 361.899,Z 567.484,A -85,B 0,C 180,E1 -13605.536,E2 -13605.536} C_VEL
LIN {X 0,Y 363.832,Z 553.893,A -85,B 0,C 180,E1 -13606.698,E2 -13606.698} C_VEL
LIN {X 0,Y 365.525,Z 539.885,A -85,B 0,C 180,E1 -13607.7,E2 -13607.7} C_VEL
LIN {X 0,Y 367.057,Z 524.632,A -85,B 0,C 180,E1 -13608.561,E2 -13608.561} C_VEL
LIN {X 0,Y 368.393,Z 508.419,A -85,B 0,C 180,E1 -13609.249,E2 -13609.249} C_VEL
LIN {X 0,Y 369.384,Z 491.794,A -85,B 0,C 180,E1 -13609.738,E2 -13609.738} C_VEL
LIN {X 0,Y 373.942,Z 342.873,A -85,B 0,C 180,E1 -13612.651,E2 -13612.651} C_VEL
LIN {X 0,Y 373.518,Z 340.962,A -85,B 0,C 180,E1 -13612.735,E2 -13612.735} C_VEL
LIN {X 0,Y 365.678,Z 324.331,A -85,B 0,C 180,E1 -13613.891,E2 -13613.891} C_VEL
LIN {X 0,Y 358.012,Z 309.528,A -85,B 0,C 180,E1 -13615.05,E2 -13615.05} C_VEL
LIN {X 0,Y 349.318,Z 295.047,A -85,B 0,C 180,E1 -13616.383,E2 -13616.383} C_VEL
LIN {X 0,Y 348.011,Z 292.646,A -85,B 0,C 180,E1 -13616.596,E2 -13616.596} C_VEL
LIN {X 0,Y 347.776,Z 291.463,A -85,B 0,C 180,E1 -13616.68,E2 -13616.68} C_VEL
LIN {X 0,Y 347.732,Z 291.486,A -85,B 0,C 180,E1 -13620.349,E2 -13620.349} C_VEL
LIN {X 0,Y 347.751,Z 291.478,A -85,B 0,C 180,E1 -13624.043,E2 -13624.043} C_VEL
LIN {X 0,Y 347.756,Z 291.478,A -85,B 0,C 180,E1 -13627.321,E2 -13627.321} C_VEL
LIN {X 0,Y 347.698,Z 291.487,A -85,B 0,C 180,E1 -13630.302,E2 -13630.302} C_VEL
LIN {X 0,Y 347.723,Z 291.48,A -85,B 0,C 180,E1 -13633.408,E2 -13633.408} C_VEL
LIN {X 0,Y 347.724,Z 291.47,A -85,B 0,C 180,E1 -13636.686,E2 -13636.686} C_VEL
LIN {X 0,Y 347.702,Z 291.478,A -85,B 0,C 180,E1 -13640.182,E2 -13640.182} C_VEL
LIN {X 0,Y 347.756,Z 291.432,A -85,B 0,C 180,E1 -13642.678,E2 -13642.678} C_VEL
LIN {X 0,Y 347.75,Z 291.461,A -85,B 0,C 180,E1 -13645.956,E2 -13645.956} C_VEL
LIN {X 0,Y 347.74,Z 291.473,A -85,B 0,C 180,E1 -13649.65,E2 -13649.65} C_VEL
LIN {X 0,Y 347.741,Z 291.483,A -85,B 0,C 180,E1 -13653.6,E2 -13653.6} C_VEL
LIN {X 0,Y 347.764,Z 291.463,A -85,B 0,C 180,E1 -13656.159,E2 -13656.159} C_VEL
LIN {X 0,Y 347.808,Z 291.471,A -85,B 0,C 180,E1 -13659.908,E2 -13659.908} C_VEL
LIN {X 0,Y 347.833,Z 291.462,A -85,B 0,C 180,E1 -13663.568,E2 -13663.568} C_VEL
LIN {X 0,Y 347.891,Z 291.452,A -85,B 0,C 180,E1 -13667.16,E2 -13667.16} C_VEL
LIN {X 0,Y 347.941,Z 291.454,A -85,B 0,C 180,E1 -13670.7,E2 -13670.7} C_VEL
LIN {X 0,Y 348.079,Z 291.431,A -85,B 0,C 180,E1 -13673.041,E2 -13673.041} C_VEL
LIN {X 0,Y 348.196,Z 291.424,A -85,B 0,C 180,E1 -13677.686,E2 -13677.686} C_VEL
LIN {X 0,Y 348.324,Z 291.39,A -85,B 0,C 180,E1 -13679.999,E2 -13679.999} C_VEL
LIN {X 0,Y 348.206,Z 291.42,A -85,B 0,C 180,E1 -13682.313,E2 -13682.313} C_VEL
LIN {X 0,Y 348.081,Z 291.414,A -85,B 0,C 180,E1 -13686.958,E2 -13686.958} C_VEL
LIN {X 0,Y 347.945,Z 291.449,A -85,B 0,C 180,E1 -13689.299,E2 -13689.299} C_VEL
LIN {X 0,Y 347.89,Z 291.458,A -85,B 0,C 180,E1 -13692.839,E2 -13692.839} C_VEL
LIN {X 0,Y 347.831,Z 291.467,A -85,B 0,C 180,E1 -13696.431,E2 -13696.431} C_VEL
LIN {X 0,Y 347.811,Z 291.473,A -85,B 0,C 180,E1 -13700.09,E2 -13700.09} C_VEL
LIN {X 0,Y 347.788,Z 291.477,A -85,B 0,C 180,E1 -13703.838,E2 -13703.838} C_VEL
LIN {X 0,Y 347.849,Z 291.469,A -85,B 0,C 180,E1 -13707.254,E2 -13707.254} C_VEL
LIN {X 0,Y 347.747,Z 291.481,A -85,B 0,C 180,E1 -13710.347,E2 -13710.347} C_VEL
LIN {X 0,Y 347.746,Z 291.48,A -85,B 0,C 180,E1 -13714.043,E2 -13714.043} C_VEL
LIN {X 0,Y 347.761,Z 291.468,A -85,B 0,C 180,E1 -13717.32,E2 -13717.32} C_VEL
LIN {X 0,Y 347.73,Z 291.474,A -85,B 0,C 180,E1 -13720.297,E2 -13720.297} C_VEL
LIN {X 0,Y 347.722,Z 291.482,A -85,B 0,C 180,E1 -13723.408,E2 -13723.408} C_VEL
LIN {X 0,Y 347.744,Z 291.477,A -85,B 0,C 180,E1 -13726.682,E2 -13726.682} C_VEL
LIN {X 0,Y 347.755,Z 291.513,A -85,B 0,C 180,E1 -13728.038,E2 -13728.038} C_VEL
LIN {X 0,Y 352.645,Z 305.772,A -85,B 0,C 180,E1 -13730.879,E2 -13730.879} C_VEL
LIN {X 0,Y 363.502,Z 327.169,A -85,B 0,C 180,E1 -13732.566,E2 -13732.566} C_VEL
LIN {X 0,Y 373.216,Z 348.421,A -85,B 0,C 180,E1 -13734.022,E2 -13734.022} C_VEL
LIN {X 0,Y 373.835,Z 353.289,A -85,B 0,C 180,E1 -13734.19,E2 -13734.19} C_VEL
LIN {X 0,Y 369.029,Z 512.983,A -85,B 0,C 180,E1 -13737.326,E2 -13737.326} C_VEL
LIN {X 0,Y 367.888,Z 529.198,A -85,B 0,C 180,E1 -13737.825,E2 -13737.825} C_VEL
LIN {X 0,Y 366.328,Z 545.965,A -85,B 0,C 180,E1 -13738.561,E2 -13738.561} C_VEL
LIN {X 0,Y 364.5,Z 562.203,A -85,B 0,C 180,E1 -13739.514,E2 -13739.514} C_VEL
LIN {X 0,Y 362.581,Z 576.271,A -85,B 0,C 180,E1 -13740.538,E2 -13740.538} C_VEL
LIN {X 0,Y 360.273,Z 591.705,A -85,B 0,C 180,E1 -13741.935,E2 -13741.935} C_VEL
LIN {X 0,Y 357.939,Z 605.657,A -85,B 0,C 180,E1 -13743.469,E2 -13743.469} C_VEL
LIN {X 0,Y 355.626,Z 618.616,A -85,B 0,C 180,E1 -13745.169,E2 -13745.169} C_VEL
LIN {X 0,Y 353.715,Z 629.782,A -85,B 0,C 180,E1 -13746.895,E2 -13746.895} C_VEL
LIN {X 0,Y 351.672,Z 640.884,A -85,B 0,C 180,E1 -13748.917,E2 -13748.917} C_VEL
LIN {X 0,Y 349.894,Z 651.594,A -85,B 0,C 180,E1 -13751.254,E2 -13751.254} C_VEL
LIN {X 0,Y 348.471,Z 660.543,A -85,B 0,C 180,E1 -13753.599,E2 -13753.599} C_VEL
LIN {X 0,Y 347.427,Z 668.595,A -85,B 0,C 180,E1 -13756.16,E2 -13756.16} C_VEL
LIN {X 0,Y 346.801,Z 674.171,A -85,B 0,C 180,E1 -13758.308,E2 -13758.308} C_VEL
LIN {X 0,Y 346.355,Z 679.057,A -85,B 0,C 180,E1 -13760.658,E2 -13760.658} C_VEL
LIN {X 0,Y 346.212,Z 682.906,A -85,B 0,C 180,E1 -13763.004,E2 -13763.004} C_VEL
LIN {X 0,Y 346.138,Z 685.602,A -85,B 0,C 180,E1 -13765.342,E2 -13765.342} C_VEL
LIN {X 0,Y 346.083,Z 687.357,A -85,B 0,C 180,E1 -13767.672,E2 -13767.672} C_VEL
LIN {X 0,Y 346.162,Z 688.06,A -85,B 0,C 180,E1 -13770,E2 -13770} C_VEL
LIN {X 0,Y 346.077,Z 687.858,A -85,B 0,C 180,E1 -13772.328,E2 -13772.328} C_VEL
LIN {X 0,Y 346.118,Z 686.618,A -85,B 0,C 180,E1 -13774.659,E2 -13774.659} C_VEL
LIN {X 0,Y 346.212,Z 684.48,A -85,B 0,C 180,E1 -13776.996,E2 -13776.996} C_VEL
LIN {X 0,Y 346.393,Z 681.267,A -85,B 0,C 180,E1 -13779.341,E2 -13779.341} C_VEL
LIN {X 0,Y 346.883,Z 677.08,A -85,B 0,C 180,E1 -13781.689,E2 -13781.689} C_VEL
LIN {X 0,Y 347.642,Z 671.75,A -85,B 0,C 180,E1 -13784.04,E2 -13784.04} C_VEL
LIN {X 0,Y 348.779,Z 665.253,A -85,B 0,C 180,E1 -13786.386,E2 -13786.386} C_VEL
LIN {X 0,Y 350.404,Z 657.497,A -85,B 0,C 180,E1 -13788.718,E2 -13788.718} C_VEL
LIN {X 0,Y 352.317,Z 648.177,A -85,B 0,C 180,E1 -13791.043,E2 -13791.043} C_VEL
LIN {X 0,Y 354.549,Z 638.609,A -85,B 0,C 180,E1 -13793.048,E2 -13793.048} C_VEL
LIN {X 0,Y 356.991,Z 628.014,A -85,B 0,C 180,E1 -13794.953,E2 -13794.953} C_VEL
LIN {X 0,Y 359.579,Z 616.43,A -85,B 0,C 180,E1 -13796.714,E2 -13796.714} C_VEL
LIN {X 0,Y 362.104,Z 604.677,A -85,B 0,C 180,E1 -13798.235,E2 -13798.235} C_VEL
LIN {X 0,Y 364.87,Z 591.5,A -85,B 0,C 180,E1 -13799.676,E2 -13799.676} C_VEL
LIN {X 0,Y 367.758,Z 576.077,A -85,B 0,C 180,E1 -13801.063,E2 -13801.063} C_VEL
LIN {X 0,Y 370.19,Z 561.512,A -85,B 0,C 180,E1 -13802.112,E2 -13802.112} C_VEL
LIN {X 0,Y 372.367,Z 545.779,A -85,B 0,C 180,E1 -13803.024,E2 -13803.024} C_VEL
LIN {X 0,Y 374.113,Z 530.637,A -85,B 0,C 180,E1 -13803.695,E2 -13803.695} C_VEL
LIN {X 0,Y 375.57,Z 513.757,A -85,B 0,C 180,E1 -13804.224,E2 -13804.224} C_VEL
LIN {X 0,Y 378.377,Z 439.185,A -85,B 0,C 180,E1 -13805.727,E2 -13805.727} C_VEL
LIN {X 0,Y 381.509,Z 354.384,A -85,B 0,C 180,E1 -13807.406,E2 -13807.406} C_VEL
LIN {X 0,Y 374.129,Z 339.5,A -85,B 0,C 180,E1 -13808.789,E2 -13808.789} C_VEL
LIN {X 0,Y 365.406,Z 324.093,A -85,B 0,C 180,E1 -13810.489,E2 -13810.489} C_VEL
LIN {X 0,Y 358.761,Z 313.268,A -85,B 0,C 180,E1 -13811.856,E2 -13811.856} C_VEL
LIN {X 0,Y 352.903,Z 304.066,A -85,B 0,C 180,E1 -13813.169,E2 -13813.169} C_VEL
LIN {X 0,Y 349.181,Z 295.028,A -85,B 0,C 180,E1 -13815.621,E2 -13815.621} C_VEL
LIN {X 0,Y 348.091,Z 292.98,A -85,B 0,C 180,E1 -13816.251,E2 -13816.251} C_VEL
LIN {X 0,Y 347.724,Z 291.484,A -85,B 0,C 180,E1 -13816.687,E2 -13816.687} C_VEL
LIN {X 0,Y 347.746,Z 291.479,A -85,B 0,C 180,E1 -13820.174,E2 -13820.174} C_VEL
LIN {X 0,Y 347.761,Z 291.46,A -85,B 0,C 180,E1 -13822.68,E2 -13822.68} C_VEL
LIN {X 0,Y 347.748,Z 291.466,A -85,B 0,C 180,E1 -13825.957,E2 -13825.957} C_VEL
LIN {X 0,Y 347.749,Z 291.48,A -85,B 0,C 180,E1 -13829.653,E2 -13829.653} C_VEL
LIN {X 0,Y 347.831,Z 291.462,A -85,B 0,C 180,E1 -13833.608,E2 -13833.608} C_VEL
LIN {X 0,Y 347.786,Z 291.456,A -85,B 0,C 180,E1 -13836.162,E2 -13836.162} C_VEL
LIN {X 0,Y 347.812,Z 291.472,A -85,B 0,C 180,E1 -13839.91,E2 -13839.91} C_VEL
LIN {X 0,Y 347.867,Z 291.44,A -85,B 0,C 180,E1 -13842.36,E2 -13842.36} C_VEL
LIN {X 0,Y 347.899,Z 291.461,A -85,B 0,C 180,E1 -13845.971,E2 -13845.971} C_VEL
LIN {X 0,Y 347.897,Z 291.429,A -85,B 0,C 180,E1 -13849.525,E2 -13849.525} C_VEL
LIN {X 0,Y 348.058,Z 291.44,A -85,B 0,C 180,E1 -13853.042,E2 -13853.042} C_VEL
LIN {X 0,Y 348.198,Z 291.417,A -85,B 0,C 180,E1 -13857.687,E2 -13857.687} C_VEL
LIN {X 0,Y 348.267,Z 291.406,A -85,B 0,C 180,E1 -13860.001,E2 -13860.001} C_VEL
LIN {X 0,Y 348.191,Z 291.394,A -85,B 0,C 180,E1 -13862.314,E2 -13862.314} C_VEL
LIN {X 0,Y 348.057,Z 291.421,A -85,B 0,C 180,E1 -13866.959,E2 -13866.959} C_VEL
LIN {X 0,Y 347.899,Z 291.46,A -85,B 0,C 180,E1 -13870.476,E2 -13870.476} C_VEL
LIN {X 0,Y 347.902,Z 291.435,A -85,B 0,C 180,E1 -13874.15,E2 -13874.15} C_VEL
LIN {X 0,Y 347.798,Z 291.454,A -85,B 0,C 180,E1 -13878.243,E2 -13878.243} C_VEL
LIN {X 0,Y 347.766,Z 291.479,A -85,B 0,C 180,E1 -13881.625,E2 -13881.625} C_VEL
LIN {X 0,Y 347.735,Z 291.47,A -85,B 0,C 180,E1 -13885.115,E2 -13885.115} C_VEL
LIN {X 0,Y 347.726,Z 291.467,A -85,B 0,C 180,E1 -13887.702,E2 -13887.702} C_VEL
LIN {X 0,Y 347.732,Z 291.485,A -85,B 0,C 180,E1 -13890.35,E2 -13890.35} C_VEL
LIN {X 0,Y 347.739,Z 291.493,A -85,B 0,C 180,E1 -13892.993,E2 -13892.993} C_VEL
LIN {X 0,Y 348.656,Z 294.183,A -85,B 0,C 180,E1 -13893.248,E2 -13893.248} C_VEL
LIN {X 0,Y 350.703,Z 296.365,A -85,B 0,C 180,E1 -13893.692,E2 -13893.692} C_VEL
LIN {X 0,Y 353.575,Z 300.559,A -85,B 0,C 180,E1 -13894.334,E2 -13894.334} C_VEL
LIN {X 0,Y 354.776,Z 302.032,A -85,B 0,C 180,E1 -13894.589,E2 -13894.589} C_VEL
LIN {X 0,Y 363.907,Z 315.017,A -85,B 0,C 180,E1 -13896.475,E2 -13896.475} C_VEL
LIN {X 0,Y 373.612,Z 331.305,A -85,B 0,C 180,E1 -13898.373,E2 -13898.373} C_VEL
LIN {X 0,Y 381.766,Z 346.552,A -85,B 0,C 180,E1 -13899.881,E2 -13899.881} C_VEL
LIN {X 0,Y 376.12,Z 494.76,A -85,B 0,C 180,E1 -13902.823,E2 -13902.823} C_VEL
LIN {X 0,Y 374.946,Z 510.748,A -85,B 0,C 180,E1 -13903.323,E2 -13903.323} C_VEL
LIN {X 0,Y 373.365,Z 526.083,A -85,B 0,C 180,E1 -13903.985,E2 -13903.985} C_VEL
LIN {X 0,Y 371.37,Z 541.883,A -85,B 0,C 180,E1 -13904.888,E2 -13904.888} C_VEL
LIN {X 0,Y 369.069,Z 556.804,A -85,B 0,C 180,E1 -13905.969,E2 -13905.969} C_VEL
LIN {X 0,Y 366.462,Z 571.448,A -85,B 0,C 180,E1 -13907.279,E2 -13907.279} C_VEL
LIN {X 0,Y 363.737,Z 585.058,A -85,B 0,C 180,E1 -13908.749,E2 -13908.749} C_VEL
LIN {X 0,Y 361.024,Z 597.767,A -85,B 0,C 180,E1 -13910.391,E2 -13910.391} C_VEL
LIN {X 0,Y 358.313,Z 609.714,A -85,B 0,C 180,E1 -13912.226,E2 -13912.226} C_VEL
LIN {X 0,Y 355.65,Z 620.644,A -85,B 0,C 180,E1 -13914.225,E2 -13914.225} C_VEL
LIN {X 0,Y 353.16,Z 631.195,A -85,B 0,C 180,E1 -13916.534,E2 -13916.534} C_VEL
LIN {X 0,Y 351.311,Z 639.349,A -85,B 0,C 180,E1 -13918.659,E2 -13918.659} C_VEL
LIN {X 0,Y 349.525,Z 647.306,A -85,B 0,C 180,E1 -13921.146,E2 -13921.146} C_VEL
LIN {X 0,Y 348.211,Z 653.714,A -85,B 0,C 180,E1 -13923.639,E2 -13923.639} C_VEL
LIN {X 0,Y 347.233,Z 658.83,A -85,B 0,C 180,E1 -13926.121,E2 -13926.121} C_VEL
LIN {X 0,Y 346.587,Z 663.126,A -85,B 0,C 180,E1 -13928.874,E2 -13928.874} C_VEL
LIN {X 0,Y 346.204,Z 665.509,A -85,B 0,C 180,E1 -13931.046,E2 -13931.046} C_VEL
LIN {X 0,Y 346.016,Z 667.241,A -85,B 0,C 180,E1 -13933.479,E2 -13933.479} C_VEL
LIN {X 0,Y 345.947,Z 667.902,A -85,B 0,C 180,E1 -13935.89,E2 -13935.89} C_VEL
LIN {X 0,Y 346.01,Z 667.593,A -85,B 0,C 180,E1 -13938.281,E2 -13938.281} C_VEL
LIN {X 0,Y 345.993,Z 666.297,A -85,B 0,C 180,E1 -13940.648,E2 -13940.648} C_VEL
LIN {X 0,Y 346.241,Z 664.011,A -85,B 0,C 180,E1 -13943.005,E2 -13943.005} C_VEL
LIN {X 0,Y 346.513,Z 660.744,A -85,B 0,C 180,E1 -13945.346,E2 -13945.346} C_VEL
LIN {X 0,Y 346.964,Z 656.401,A -85,B 0,C 180,E1 -13947.678,E2 -13947.678} C_VEL
LIN {X 0,Y 347.582,Z 651.035,A -85,B 0,C 180,E1 -13950,E2 -13950} C_VEL
LIN {X 0,Y 348.577,Z 644.372,A -85,B 0,C 180,E1 -13952.311,E2 -13952.311} C_VEL
LIN {X 0,Y 349.856,Z 636.426,A -85,B 0,C 180,E1 -13954.609,E2 -13954.609} C_VEL
LIN {X 0,Y 351.638,Z 626.965,A -85,B 0,C 180,E1 -13956.887,E2 -13956.887} C_VEL
LIN {X 0,Y 353.478,Z 617.204,A -85,B 0,C 180,E1 -13958.864,E2 -13958.864} C_VEL
LIN {X 0,Y 355.517,Z 605.791,A -85,B 0,C 180,E1 -13960.824,E2 -13960.824} C_VEL
LIN {X 0,Y 357.658,Z 593.385,A -85,B 0,C 180,E1 -13962.627,E2 -13962.627} C_VEL
LIN {X 0,Y 359.889,Z 579.9,A -85,B 0,C 180,E1 -13964.273,E2 -13964.273} C_VEL
LIN {X 0,Y 361.899,Z 567.484,A -85,B 0,C 180,E1 -13965.536,E2 -13965.536} C_VEL
LIN {X 0,Y 362.027,Z 562.511,A -85,B 0,C 180,E1 -13966.043,E2 -13966.043} C_VEL
LIN {X 0,Y 359.237,Z 547.823,A -85,B 0,C 180,E1 -13967.599,E2 -13967.599} C_VEL
LIN {X 0,Y 358.963,Z 542.613,A -85,B 0,C 180,E1 -13968.038,E2 -13968.038} C_VEL
LIN {X 0,Y 359.136,Z 540.823,A -85,B 0,C 180,E1 -13968.165,E2 -13968.165} C_VEL
LIN {X 0,Y 360.722,Z 525.57,A -85,B 0,C 180,E1 -13969.047,E2 -13969.047} C_VEL
LIN {X 0,Y 362.093,Z 509.644,A -85,B 0,C 180,E1 -13969.746,E2 -13969.746} C_VEL
LIN {X 0,Y 363.131,Z 493.631,A -85,B 0,C 180,E1 -13970.24,E2 -13970.24} C_VEL
LIN {X 0,Y 367.932,Z 344.204,A -85,B 0,C 180,E1 -13973.207,E2 -13973.207} C_VEL
LIN {X 0,Y 360.412,Z 328.172,A -85,B 0,C 180,E1 -13974.349,E2 -13974.349} C_VEL
LIN {X 0,Y 353.199,Z 314.044,A -85,B 0,C 180,E1 -13975.473,E2 -13975.473} C_VEL
LIN {X 0,Y 342.412,Z 296.133,A -85,B 0,C 180,E1 -13977.179,E2 -13977.179} C_VEL
LIN {X 0,Y 340.944,Z 293.511,A -85,B 0,C 180,E1 -13977.427,E2 -13977.427} C_VEL
LIN {X 0,Y 340.692,Z 292.357,A -85,B 0,C 180,E1 -13977.496,E2 -13977.496} C_VEL
LIN {X 0,Y 340.685,Z 292.364,A -85,B 0,C 180,E1 -13981.046,E2 -13981.046} C_VEL
LIN {X 0,Y 340.718,Z 292.348,A -85,B 0,C 180,E1 -13985.279,E2 -13985.279} C_VEL
LIN {X 0,Y 340.695,Z 292.351,A -85,B 0,C 180,E1 -13988.382,E2 -13988.382} C_VEL
LIN {X 0,Y 340.692,Z 292.349,A -85,B 0,C 180,E1 -13992.043,E2 -13992.043} C_VEL
LIN {X 0,Y 340.651,Z 292.351,A -85,B 0,C 180,E1 -13996.227,E2 -13996.227} C_VEL
LIN {X 0,Y 340.67,Z 292.362,A -85,B 0,C 180,E1 -13998.687,E2 -13998.687} C_VEL
LIN {X 0,Y 340.72,Z 292.321,A -85,B 0,C 180,E1 -14001.77,E2 -14001.77} C_VEL
LIN {X 0,Y 340.724,Z 292.331,A -85,B 0,C 180,E1 -14005.595,E2 -14005.595} C_VEL
LIN {X 0,Y 340.695,Z 292.357,A -85,B 0,C 180,E1 -14008.954,E2 -14008.954} C_VEL
LIN {X 0,Y 340.713,Z 292.354,A -85,B 0,C 180,E1 -14013.011,E2 -14013.011} C_VEL
LIN {X 0,Y 340.74,Z 292.34,A -85,B 0,C 180,E1 -14015.636,E2 -14015.636} C_VEL
LIN {X 0,Y 340.736,Z 292.356,A -85,B 0,C 180,E1 -14019.473,E2 -14019.473} C_VEL
LIN {X 0,Y 340.794,Z 292.33,A -85,B 0,C 180,E1 -14021.98,E2 -14021.98} C_VEL
LIN {X 0,Y 340.871,Z 292.336,A -85,B 0,C 180,E1 -14025.704,E2 -14025.704} C_VEL
LIN {X 0,Y 340.871,Z 292.325,A -85,B 0,C 180,E1 -14029.306,E2 -14029.306} C_VEL
LIN {X 0,Y 341.046,Z 292.309,A -85,B 0,C 180,E1 -14032.897,E2 -14032.897} C_VEL
LIN {X 0,Y 341.157,Z 292.302,A -85,B 0,C 180,E1 -14037.638,E2 -14037.638} C_VEL
LIN {X 0,Y 341.275,Z 292.268,A -85,B 0,C 180,E1 -14039.999,E2 -14039.999} C_VEL
LIN {X 0,Y 341.168,Z 292.297,A -85,B 0,C 180,E1 -14042.361,E2 -14042.361} C_VEL
LIN {X 0,Y 341.051,Z 292.289,A -85,B 0,C 180,E1 -14047.102,E2 -14047.102} C_VEL
LIN {X 0,Y 340.871,Z 292.337,A -85,B 0,C 180,E1 -14050.693,E2 -14050.693} C_VEL
LIN {X 0,Y 340.862,Z 292.338,A -85,B 0,C 180,E1 -14054.324,E2 -14054.324} C_VEL
LIN {X 0,Y 340.785,Z 292.348,A -85,B 0,C 180,E1 -14058.44,E2 -14058.44} C_VEL
LIN {X 0,Y 340.753,Z 292.349,A -85,B 0,C 180,E1 -14061.856,E2 -14061.856} C_VEL
LIN {X 0,Y 340.771,Z 292.35,A -85,B 0,C 180,E1 -14065.664,E2 -14065.664} C_VEL
LIN {X 0,Y 340.727,Z 292.351,A -85,B 0,C 180,E1 -14068.32,E2 -14068.32} C_VEL
LIN {X 0,Y 340.696,Z 292.358,A -85,B 0,C 180,E1 -14071.044,E2 -14071.044} C_VEL
LIN {X 0,Y 340.717,Z 292.352,A -85,B 0,C 180,E1 -14075.278,E2 -14075.278} C_VEL
LIN {X 0,Y 340.708,Z 292.357,A -85,B 0,C 180,E1 -14078.386,E2 -14078.386} C_VEL
LIN {X 0,Y 340.697,Z 292.358,A -85,B 0,C 180,E1 -14082.045,E2 -14082.045} C_VEL
LIN {X 0,Y 340.689,Z 292.359,A -85,B 0,C 180,E1 -14085.462,E2 -14085.462} C_VEL
LIN {X 0,Y 340.73,Z 292.466,A -85,B 0,C 180,E1 -14087.324,E2 -14087.324} C_VEL
LIN {X 0,Y 345.327,Z 305.639,A -85,B 0,C 180,E1 -14090.028,E2 -14090.028} C_VEL
LIN {X 0,Y 356.476,Z 327.312,A -85,B 0,C 180,E1 -14091.826,E2 -14091.826} C_VEL
LIN {X 0,Y 366.771,Z 349.521,A -85,B 0,C 180,E1 -14093.417,E2 -14093.417} C_VEL
LIN {X 0,Y 367.503,Z 351.56,A -85,B 0,C 180,E1 -14093.536,E2 -14093.536} C_VEL
LIN {X 0,Y 367.752,Z 355.324,A -85,B 0,C 180,E1 -14093.647,E2 -14093.647} C_VEL
LIN {X 0,Y 362.791,Z 513.563,A -85,B 0,C 180,E1 -14096.801,E2 -14096.801} C_VEL
LIN {X 0,Y 361.534,Z 530.757,A -85,B 0,C 180,E1 -14097.354,E2 -14097.354} C_VEL
LIN {X 0,Y 359.923,Z 547.026,A -85,B 0,C 180,E1 -14098.1,E2 -14098.1} C_VEL
LIN {X 0,Y 358.037,Z 562.978,A -85,B 0,C 180,E1 -14099.067,E2 -14099.067} C_VEL
LIN {X 0,Y 356.055,Z 576.873,A -85,B 0,C 180,E1 -14100.106,E2 -14100.106} C_VEL
LIN {X 0,Y 353.693,Z 592.131,A -85,B 0,C 180,E1 -14101.518,E2 -14101.518} C_VEL
LIN {X 0,Y 351.26,Z 606.04,A -85,B 0,C 180,E1 -14103.084,E2 -14103.084} C_VEL
LIN {X 0,Y 349.074,Z 617.907,A -85,B 0,C 180,E1 -14104.67,E2 -14104.67} C_VEL
LIN {X 0,Y 347.061,Z 629.154,A -85,B 0,C 180,E1 -14106.426,E2 -14106.426} C_VEL
LIN {X 0,Y 344.918,Z 640.294,A -85,B 0,C 180,E1 -14108.484,E2 -14108.484} C_VEL
LIN {X 0,Y 343.07,Z 651.072,A -85,B 0,C 180,E1 -14110.867,E2 -14110.867} C_VEL
LIN {X 0,Y 341.527,Z 660.083,A -85,B 0,C 180,E1 -14113.256,E2 -14113.256} C_VEL
LIN {X 0,Y 340.504,Z 667.619,A -85,B 0,C 180,E1 -14115.66,E2 -14115.66} C_VEL
LIN {X 0,Y 339.776,Z 673.797,A -85,B 0,C 180,E1 -14118.063,E2 -14118.063} C_VEL
LIN {X 0,Y 339.283,Z 678.724,A -85,B 0,C 180,E1 -14120.461,E2 -14120.461} C_VEL
LIN {X 0,Y 339.125,Z 682.608,A -85,B 0,C 180,E1 -14122.857,E2 -14122.857} C_VEL
LIN {X 0,Y 339.041,Z 685.329,A -85,B 0,C 180,E1 -14125.244,E2 -14125.244} C_VEL
LIN {X 0,Y 338.997,Z 687.122,A -85,B 0,C 180,E1 -14127.624,E2 -14127.624} C_VEL
LIN {X 0,Y 339.065,Z 687.843,A -85,B 0,C 180,E1 -14130,E2 -14130} C_VEL
LIN {X 0,Y 338.991,Z 687.676,A -85,B 0,C 180,E1 -14132.377,E2 -14132.377} C_VEL
LIN {X 0,Y 339.021,Z 686.454,A -85,B 0,C 180,E1 -14134.757,E2 -14134.757} C_VEL
LIN {X 0,Y 339.126,Z 684.352,A -85,B 0,C 180,E1 -14137.143,E2 -14137.143} C_VEL
LIN {X 0,Y 339.321,Z 681.162,A -85,B 0,C 180,E1 -14139.538,E2 -14139.538} C_VEL
LIN {X 0,Y 339.872,Z 677.021,A -85,B 0,C 180,E1 -14141.934,E2 -14141.934} C_VEL
LIN {X 0,Y 340.66,Z 671.715,A -85,B 0,C 180,E1 -14144.334,E2 -14144.334} C_VEL
LIN {X 0,Y 341.876,Z 665.265,A -85,B 0,C 180,E1 -14146.726,E2 -14146.726} C_VEL
LIN {X 0,Y 343.586,Z 657.547,A -85,B 0,C 180,E1 -14149.104,E2 -14149.104} C_VEL
LIN {X 0,Y 345.628,Z 648.275,A -85,B 0,C 180,E1 -14151.47,E2 -14151.47} C_VEL
LIN {X 0,Y 347.96,Z 638.783,A -85,B 0,C 180,E1 -14153.51,E2 -14153.51} C_VEL
LIN {X 0,Y 350.71,Z 627.285,A -85,B 0,C 180,E1 -14155.609,E2 -14155.609} C_VEL
LIN {X 0,Y 353.691,Z 614.795,A -85,B 0,C 180,E1 -14157.516,E2 -14157.516} C_VEL
LIN {X 0,Y 356.155,Z 603.919,A -85,B 0,C 180,E1 -14158.912,E2 -14158.912} C_VEL
LIN {X 0,Y 359.064,Z 590.263,A -85,B 0,C 180,E1 -14160.41,E2 -14160.41} C_VEL
LIN {X 0,Y 362.024,Z 575.088,A -85,B 0,C 180,E1 -14161.775,E2 -14161.775} C_VEL
LIN {X 0,Y 364.877,Z 558.426,A -85,B 0,C 180,E1 -14162.965,E2 -14162.965} C_VEL
LIN {X 0,Y 367.146,Z 541.861,A -85,B 0,C 180,E1 -14163.885,E2 -14163.885} C_VEL
LIN {X 0,Y 369.027,Z 525.217,A -85,B 0,C 180,E1 -14164.554,E2 -14164.554} C_VEL
LIN {X 0,Y 370.279,Z 508.693,A -85,B 0,C 180,E1 -14165.015,E2 -14165.015} C_VEL
LIN {X 0,Y 376.143,Z 356.929,A -85,B 0,C 180,E1 -14168.062,E2 -14168.062} C_VEL
LIN {X 0,Y 369.135,Z 342.856,A -85,B 0,C 180,E1 -14169.421,E2 -14169.421} C_VEL
LIN {X 0,Y 361.039,Z 328.486,A -85,B 0,C 180,E1 -14171.054,E2 -14171.054} C_VEL
LIN {X 0,Y 354.91,Z 318.382,A -85,B 0,C 180,E1 -14172.356,E2 -14172.356} C_VEL
LIN {X 0,Y 348.142,Z 308.016,A -85,B 0,C 180,E1 -14173.869,E2 -14173.869} C_VEL
LIN {X 0,Y 345.335,Z 303.683,A -85,B 0,C 180,E1 -14174.579,E2 -14174.579} C_VEL
LIN {X 0,Y 342.036,Z 295.718,A -85,B 0,C 180,E1 -14176.872,E2 -14176.872} C_VEL
LIN {X 0,Y 340.898,Z 293.382,A -85,B 0,C 180,E1 -14177.609,E2 -14177.609} C_VEL
LIN {X 0,Y 340.698,Z 292.344,A -85,B 0,C 180,E1 -14177.955,E2 -14177.955} C_VEL
LIN {X 0,Y 340.732,Z 292.339,A -85,B 0,C 180,E1 -14181.773,E2 -14181.773} C_VEL
LIN {X 0,Y 340.722,Z 292.346,A -85,B 0,C 180,E1 -14185.596,E2 -14185.596} C_VEL
LIN {X 0,Y 340.698,Z 292.356,A -85,B 0,C 180,E1 -14188.956,E2 -14188.956} C_VEL
LIN {X 0,Y 340.803,Z 292.325,A -85,B 0,C 180,E1 -14193.021,E2 -14193.021} C_VEL
LIN {X 0,Y 340.755,Z 292.341,A -85,B 0,C 180,E1 -14195.639,E2 -14195.639} C_VEL
LIN {X 0,Y 340.739,Z 292.35,A -85,B 0,C 180,E1 -14199.474,E2 -14199.474} C_VEL
LIN {X 0,Y 340.859,Z 292.317,A -85,B 0,C 180,E1 -14201.985,E2 -14201.985} C_VEL
LIN {X 0,Y 340.87,Z 292.336,A -85,B 0,C 180,E1 -14205.706,E2 -14205.706} C_VEL
LIN {X 0,Y 340.849,Z 292.306,A -85,B 0,C 180,E1 -14209.306,E2 -14209.306} C_VEL
LIN {X 0,Y 341.004,Z 292.319,A -85,B 0,C 180,E1 -14212.897,E2 -14212.897} C_VEL
LIN {X 0,Y 340.828,Z 292.308,A -85,B 0,C 180,E1 -14215.269,E2 -14215.269} C_VEL
LIN {X 0,Y 341.159,Z 292.291,A -85,B 0,C 180,E1 -14217.639,E2 -14217.639} C_VEL
LIN {X 0,Y 341.219,Z 292.283,A -85,B 0,C 180,E1 -14220.001,E2 -14220.001} C_VEL
LIN {X 0,Y 341.128,Z 292.273,A -85,B 0,C 180,E1 -14222.362,E2 -14222.362} C_VEL
LIN {X 0,Y 340.993,Z 292.305,A -85,B 0,C 180,E1 -14226.542,E2 -14226.542} C_VEL
LIN {X 0,Y 340.884,Z 292.318,A -85,B 0,C 180,E1 -14229.494,E2 -14229.494} C_VEL
LIN {X 0,Y 340.846,Z 292.316,A -85,B 0,C 180,E1 -14233.11,E2 -14233.11} C_VEL
LIN {X 0,Y 340.801,Z 292.336,A -85,B 0,C 180,E1 -14235.551,E2 -14235.551} C_VEL
LIN {X 0,Y 340.711,Z 292.331,A -85,B 0,C 180,E1 -14239.272,E2 -14239.272} C_VEL
LIN {X 0,Y 340.702,Z 292.342,A -85,B 0,C 180,E1 -14243.076,E2 -14243.076} C_VEL
LIN {X 0,Y 340.712,Z 292.348,A -85,B 0,C 180,E1 -14246.989,E2 -14246.989} C_VEL
LIN {X 0,Y 340.719,Z 292.356,A -85,B 0,C 180,E1 -14249.964,E2 -14249.964} C_VEL
LIN {X 0,Y 340.719,Z 292.535,A -85,B 0,C 180,E1 -14251.649,E2 -14251.649} C_VEL
LIN {X 0,Y 341.557,Z 294.979,A -85,B 0,C 180,E1 -14251.898,E2 -14251.898} C_VEL
LIN {X 0,Y 343.489,Z 297.128,A -85,B 0,C 180,E1 -14252.352,E2 -14252.352} C_VEL
LIN {X 0,Y 344.3,Z 297.941,A -85,B 0,C 180,E1 -14252.537,E2 -14252.537} C_VEL
LIN {X 0,Y 346.269,Z 301.097,A -85,B 0,C 180,E1 -14253.014,E2 -14253.014} C_VEL
LIN {X 0,Y 347.922,Z 302.977,A -85,B 0,C 180,E1 -14253.382,E2 -14253.382} C_VEL
LIN {X 0,Y 350.508,Z 306.547,A -85,B 0,C 180,E1 -14253.966,E2 -14253.966} C_VEL
LIN {X 0,Y 359.975,Z 320.02,A -85,B 0,C 180,E1 -14255.983,E2 -14255.983} C_VEL
LIN {X 0,Y 369.284,Z 335.883,A -85,B 0,C 180,E1 -14257.863,E2 -14257.863} C_VEL
LIN {X 0,Y 376.378,Z 349.221,A -85,B 0,C 180,E1 -14259.222,E2 -14259.222} C_VEL
LIN {X 0,Y 370.544,Z 495.661,A -85,B 0,C 180,E1 -14262.162,E2 -14262.162} C_VEL
LIN {X 0,Y 369.269,Z 511.884,A -85,B 0,C 180,E1 -14262.683,E2 -14262.683} C_VEL
LIN {X 0,Y 367.538,Z 527.762,A -85,B 0,C 180,E1 -14263.395,E2 -14263.395} C_VEL
LIN {X 0,Y 365.439,Z 543.225,A -85,B 0,C 180,E1 -14264.306,E2 -14264.306} C_VEL
LIN {X 0,Y 363.022,Z 558.314,A -85,B 0,C 180,E1 -14265.429,E2 -14265.429} C_VEL
LIN {X 0,Y 360.275,Z 572.947,A -85,B 0,C 180,E1 -14266.778,E2 -14266.778} C_VEL
LIN {X 0,Y 357.518,Z 586.073,A -85,B 0,C 180,E1 -14268.238,E2 -14268.238} C_VEL
LIN {X 0,Y 354.403,Z 599.72,A -85,B 0,C 180,E1 -14270.058,E2 -14270.058} C_VEL
LIN {X 0,Y 351.425,Z 612.129,A -85,B 0,C 180,E1 -14272.051,E2 -14272.051} C_VEL
LIN {X 0,Y 348.624,Z 623.418,A -85,B 0,C 180,E1 -14274.224,E2 -14274.224} C_VEL
LIN {X 0,Y 346.314,Z 632.497,A -85,B 0,C 180,E1 -14276.31,E2 -14276.31} C_VEL
LIN {X 0,Y 344.258,Z 640.963,A -85,B 0,C 180,E1 -14278.629,E2 -14278.629} C_VEL
LIN {X 0,Y 342.443,Z 648.647,A -85,B 0,C 180,E1 -14281.165,E2 -14281.165} C_VEL
LIN {X 0,Y 341.118,Z 654.905,A -85,B 0,C 180,E1 -14283.707,E2 -14283.707} C_VEL
LIN {X 0,Y 340.135,Z 659.773,A -85,B 0,C 180,E1 -14286.239,E2 -14286.239} C_VEL
LIN {X 0,Y 339.539,Z 663.377,A -85,B 0,C 180,E1 -14288.662,E2 -14288.662} C_VEL
LIN {X 0,Y 339.181,Z 665.527,A -85,B 0,C 180,E1 -14290.638,E2 -14290.638} C_VEL
LIN {X 0,Y 338.96,Z 667.365,A -85,B 0,C 180,E1 -14293.125,E2 -14293.125} C_VEL
LIN {X 0,Y 338.856,Z 668.085,A -85,B 0,C 180,E1 -14295.588,E2 -14295.588} C_VEL
LIN {X 0,Y 338.918,Z 667.885,A -85,B 0,C 180,E1 -14298.032,E2 -14298.032} C_VEL
LIN {X 0,Y 338.885,Z 666.643,A -85,B 0,C 180,E1 -14300.45,E2 -14300.45} C_VEL
LIN {X 0,Y 339.127,Z 664.466,A -85,B 0,C 180,E1 -14302.857,E2 -14302.857} C_VEL
LIN {X 0,Y 339.428,Z 661.251,A -85,B 0,C 180,E1 -14305.249,E2 -14305.249} C_VEL
LIN {X 0,Y 339.875,Z 657.022,A -85,B 0,C 180,E1 -14307.63,E2 -14307.63} C_VEL
LIN {X 0,Y 340.489,Z 651.719,A -85,B 0,C 180,E1 -14310,E2 -14310} C_VEL
LIN {X 0,Y 341.53,Z 645.169,A -85,B 0,C 180,E1 -14312.359,E2 -14312.359} C_VEL
LIN {X 0,Y 342.817,Z 637.361,A -85,B 0,C 180,E1 -14314.704,E2 -14314.704} C_VEL
LIN {X 0,Y 344.649,Z 628.043,A -85,B 0,C 180,E1 -14317.028,E2 -14317.028} C_VEL
LIN {X 0,Y 346.817,Z 616.915,A -85,B 0,C 180,E1 -14319.33,E2 -14319.33} C_VEL
LIN {X 0,Y 348.961,Z 605.401,A -85,B 0,C 180,E1 -14321.324,E2 -14321.324} C_VEL
LIN {X 0,Y 351.223,Z 592.872,A -85,B 0,C 180,E1 -14323.157,E2 -14323.157} C_VEL
LIN {X 0,Y 353.535,Z 579.241,A -85,B 0,C 180,E1 -14324.829,E2 -14324.829} C_VEL
LIN {X 0,Y 355.778,Z 565.78,A -85,B 0,C 180,E1 -14326.202,E2 -14326.202} C_VEL
LIN {X 0,Y 357.859,Z 551.164,A -85,B 0,C 180,E1 -14327.427,E2 -14327.427} C_VEL
LIN {X 0,Y 359.136,Z 540.823,A -85,B 0,C 180,E1 -14328.165,E2 -14328.165} C_VEL
LIN {X 0,Y 359.258,Z 535.454,A -85,B 0,C 180,E1 -14328.559,E2 -14328.559} C_VEL
LIN {X 0,Y 357.628,Z 526.747,A -85,B 0,C 180,E1 -14329.279,E2 -14329.279} C_VEL
LIN {X 0,Y 355.849,Z 517.864,A -85,B 0,C 180,E1 -14329.928,E2 -14329.928} C_VEL
LIN {X 0,Y 355.719,Z 512.222,A -85,B 0,C 180,E1 -14330.208,E2 -14330.208} C_VEL
LIN {X 0,Y 356.904,Z 495.465,A -85,B 0,C 180,E1 -14330.76,E2 -14330.76} C_VEL
LIN {X 0,Y 361.415,Z 359.866,A -85,B 0,C 180,E1 -14333.5,E2 -14333.5} C_VEL
LIN {X 0,Y 361.734,Z 345.882,A -85,B 0,C 180,E1 -14333.794,E2 -14333.794} C_VEL
LIN {X 0,Y 352.839,Z 327.15,A -85,B 0,C 180,E1 -14335.193,E2 -14335.193} C_VEL
LIN {X 0,Y 347.766,Z 317.52,A -85,B 0,C 180,E1 -14336.003,E2 -14336.003} C_VEL
LIN {X 0,Y 337.625,Z 300.653,A -85,B 0,C 180,E1 -14337.656,E2 -14337.656} C_VEL
LIN {X 0,Y 335.629,Z 297.357,A -85,B 0,C 180,E1 -14337.997,E2 -14337.997} C_VEL
LIN {X 0,Y 334.037,Z 294.848,A -85,B 0,C 180,E1 -14338.269,E2 -14338.269} C_VEL
LIN {X 0,Y 333.634,Z 293.245,A -85,B 0,C 180,E1 -14338.376,E2 -14338.376} C_VEL
LIN {X 0,Y 333.623,Z 293.237,A -85,B 0,C 180,E1 -14341.779,E2 -14341.779} C_VEL
LIN {X 0,Y 333.687,Z 293.224,A -85,B 0,C 180,E1 -14344.773,E2 -14344.773} C_VEL
LIN {X 0,Y 333.645,Z 293.231,A -85,B 0,C 180,E1 -14347.652,E2 -14347.652} C_VEL
LIN {X 0,Y 333.605,Z 293.24,A -85,B 0,C 180,E1 -14350.773,E2 -14350.773} C_VEL
LIN {X 0,Y 333.592,Z 293.245,A -85,B 0,C 180,E1 -14354.249,E2 -14354.249} C_VEL
LIN {X 0,Y 333.637,Z 293.23,A -85,B 0,C 180,E1 -14357.617,E2 -14357.617} C_VEL
LIN {X 0,Y 333.617,Z 293.214,A -85,B 0,C 180,E1 -14361.21,E2 -14361.21} C_VEL
LIN {X 0,Y 333.674,Z 293.182,A -85,B 0,C 180,E1 -14363.86,E2 -14363.86} C_VEL
LIN {X 0,Y 333.645,Z 293.233,A -85,B 0,C 180,E1 -14367.412,E2 -14367.412} C_VEL
LIN {X 0,Y 333.633,Z 293.222,A -85,B 0,C 180,E1 -14371.02,E2 -14371.02} C_VEL
LIN {X 0,Y 333.696,Z 293.224,A -85,B 0,C 180,E1 -14375.087,E2 -14375.087} C_VEL
LIN {X 0,Y 333.668,Z 293.233,A -85,B 0,C 180,E1 -14379.018,E2 -14379.018} C_VEL
LIN {X 0,Y 333.743,Z 293.21,A -85,B 0,C 180,E1 -14381.586,E2 -14381.586} C_VEL
LIN {X 0,Y 333.81,Z 293.217,A -85,B 0,C 180,E1 -14385.576,E2 -14385.576} C_VEL
LIN {X 0,Y 333.834,Z 293.199,A -85,B 0,C 180,E1 -14389.077,E2 -14389.077} C_VEL
LIN {X 0,Y 333.993,Z 293.189,A -85,B 0,C 180,E1 -14392.746,E2 -14392.746} C_VEL
LIN {X 0,Y 333.796,Z 293.203,A -85,B 0,C 180,E1 -14395.168,E2 -14395.168} C_VEL
LIN {X 0,Y 334.094,Z 293.182,A -85,B 0,C 180,E1 -14397.588,E2 -14397.588} C_VEL
LIN {X 0,Y 334.226,Z 293.145,A -85,B 0,C 180,E1 -14399.999,E2 -14399.999} C_VEL
LIN {X 0,Y 334.105,Z 293.176,A -85,B 0,C 180,E1 -14402.411,E2 -14402.411} C_VEL
LIN {X 0,Y 334.007,Z 293.173,A -85,B 0,C 180,E1 -14406.038,E2 -14406.038} C_VEL
LIN {X 0,Y 333.97,Z 293.182,A -85,B 0,C 180,E1 -14408.484,E2 -14408.484} C_VEL
LIN {X 0,Y 333.791,Z 293.213,A -85,B 0,C 180,E1 -14412.154,E2 -14412.154} C_VEL
LIN {X 0,Y 333.808,Z 293.218,A -85,B 0,C 180,E1 -14414.634,E2 -14414.634} C_VEL
LIN {X 0,Y 333.752,Z 293.224,A -85,B 0,C 180,E1 -14418.633,E2 -14418.633} C_VEL
LIN {X 0,Y 333.691,Z 293.228,A -85,B 0,C 180,E1 -14422.278,E2 -14422.278} C_VEL
LIN {X 0,Y 333.734,Z 293.227,A -85,B 0,C 180,E1 -14426.246,E2 -14426.246} C_VEL
LIN {X 0,Y 333.689,Z 293.233,A -85,B 0,C 180,E1 -14428.974,E2 -14428.974} C_VEL
LIN {X 0,Y 333.642,Z 293.239,A -85,B 0,C 180,E1 -14432.586,E2 -14432.586} C_VEL
LIN {X 0,Y 333.675,Z 293.221,A -85,B 0,C 180,E1 -14436.138,E2 -14436.138} C_VEL
LIN {X 0,Y 333.645,Z 293.238,A -85,B 0,C 180,E1 -14439.192,E2 -14439.192} C_VEL
LIN {X 0,Y 333.631,Z 293.242,A -85,B 0,C 180,E1 -14442.5,E2 -14442.5} C_VEL
LIN {X 0,Y 333.684,Z 293.354,A -85,B 0,C 180,E1 -14446.564,E2 -14446.564} C_VEL
LIN {X 0,Y 337.961,Z 305.397,A -85,B 0,C 180,E1 -14449.125,E2 -14449.125} C_VEL
LIN {X 0,Y 349.089,Z 326.646,A -85,B 0,C 180,E1 -14450.991,E2 -14450.991} C_VEL
LIN {X 0,Y 359.039,Z 347.849,A -85,B 0,C 180,E1 -14452.588,E2 -14452.588} C_VEL
LIN {X 0,Y 361.777,Z 354.421,A -85,B 0,C 180,E1 -14453.025,E2 -14453.025} C_VEL
LIN {X 0,Y 356.626,Z 513.405,A -85,B 0,C 180,E1 -14456.244,E2 -14456.244} C_VEL
LIN {X 0,Y 355.319,Z 530.394,A -85,B 0,C 180,E1 -14456.795,E2 -14456.795} C_VEL
LIN {X 0,Y 353.671,Z 546.711,A -85,B 0,C 180,E1 -14457.552,E2 -14457.552} C_VEL
LIN {X 0,Y 351.734,Z 562.69,A -85,B 0,C 180,E1 -14458.533,E2 -14458.533} C_VEL
LIN {X 0,Y 349.546,Z 577.405,A -85,B 0,C 180,E1 -14459.658,E2 -14459.658} C_VEL
LIN {X 0,Y 347.343,Z 591.148,A -85,B 0,C 180,E1 -14460.948,E2 -14460.948} C_VEL
LIN {X 0,Y 345.025,Z 604.007,A -85,B 0,C 180,E1 -14462.393,E2 -14462.393} C_VEL
LIN {X 0,Y 342.962,Z 615.199,A -85,B 0,C 180,E1 -14463.859,E2 -14463.859} C_VEL
LIN {X 0,Y 340.763,Z 626.696,A -85,B 0,C 180,E1 -14465.639,E2 -14465.639} C_VEL
LIN {X 0,Y 338.511,Z 638.191,A -85,B 0,C 180,E1 -14467.735,E2 -14467.735} C_VEL
LIN {X 0,Y 336.526,Z 648.698,A -85,B 0,C 180,E1 -14470.013,E2 -14470.013} C_VEL
LIN {X 0,Y 335.023,Z 657.556,A -85,B 0,C 180,E1 -14472.292,E2 -14472.292} C_VEL
LIN {X 0,Y 333.742,Z 665.43,A -85,B 0,C 180,E1 -14474.738,E2 -14474.738} C_VEL
LIN {X 0,Y 332.906,Z 671.956,A -85,B 0,C 180,E1 -14477.193,E2 -14477.193} C_VEL
LIN {X 0,Y 332.273,Z 677.288,A -85,B 0,C 180,E1 -14479.643,E2 -14479.643} C_VEL
LIN {X 0,Y 332.026,Z 682.297,A -85,B 0,C 180,E1 -14482.704,E2 -14482.704} C_VEL
LIN {X 0,Y 331.948,Z 685.054,A -85,B 0,C 180,E1 -14485.142,E2 -14485.142} C_VEL
LIN {X 0,Y 331.913,Z 686.88,A -85,B 0,C 180,E1 -14487.573,E2 -14487.573} C_VEL
LIN {X 0,Y 331.968,Z 687.626,A -85,B 0,C 180,E1 -14490,E2 -14490} C_VEL
LIN {X 0,Y 331.907,Z 687.488,A -85,B 0,C 180,E1 -14492.427,E2 -14492.427} C_VEL
LIN {X 0,Y 331.93,Z 686.294,A -85,B 0,C 180,E1 -14494.859,E2 -14494.859} C_VEL
LIN {X 0,Y 332.028,Z 684.222,A -85,B 0,C 180,E1 -14497.297,E2 -14497.297} C_VEL
LIN {X 0,Y 332.264,Z 681.063,A -85,B 0,C 180,E1 -14499.742,E2 -14499.742} C_VEL
LIN {X 0,Y 332.868,Z 676.963,A -85,B 0,C 180,E1 -14502.189,E2 -14502.189} C_VEL
LIN {X 0,Y 333.948,Z 670.237,A -85,B 0,C 180,E1 -14505.252,E2 -14505.252} C_VEL
LIN {X 0,Y 335.855,Z 661.629,A -85,B 0,C 180,E1 -14508.294,E2 -14508.294} C_VEL
LIN {X 0,Y 338.086,Z 652.065,A -85,B 0,C 180,E1 -14511.014,E2 -14511.014} C_VEL
LIN {X 0,Y 340.699,Z 641.823,A -85,B 0,C 180,E1 -14513.397,E2 -14513.397} C_VEL
LIN {X 0,Y 343.363,Z 631.284,A -85,B 0,C 180,E1 -14515.457,E2 -14515.457} C_VEL
LIN {X 0,Y 346.423,Z 618.974,A -85,B 0,C 180,E1 -14517.486,E2 -14517.486} C_VEL
LIN {X 0,Y 349.409,Z 606.665,A -85,B 0,C 180,E1 -14519.194,E2 -14519.194} C_VEL
LIN {X 0,Y 352.463,Z 593.287,A -85,B 0,C 180,E1 -14520.733,E2 -14520.733} C_VEL
LIN {X 0,Y 355.448,Z 578.937,A -85,B 0,C 180,E1 -14522.099,E2 -14522.099} C_VEL
LIN {X 0,Y 358.369,Z 563.252,A -85,B 0,C 180,E1 -14523.306,E2 -14523.306} C_VEL
LIN {X 0,Y 360.709,Z 548.201,A -85,B 0,C 180,E1 -14524.236,E2 -14524.236} C_VEL
LIN {X 0,Y 362.528,Z 533.782,A -85,B 0,C 180,E1 -14524.925,E2 -14524.925} C_VEL
LIN {X 0,Y 364.193,Z 516.975,A -85,B 0,C 180,E1 -14525.504,E2 -14525.504} C_VEL
LIN {X 0,Y 365.363,Z 495.453,A -85,B 0,C 180,E1 -14525.993,E2 -14525.993} C_VEL
LIN {X 0,Y 370.745,Z 359.412,A -85,B 0,C 180,E1 -14528.752,E2 -14528.752} C_VEL
LIN {X 0,Y 364.395,Z 346.599,A -85,B 0,C 180,E1 -14530.031,E2 -14530.031} C_VEL
LIN {X 0,Y 356.844,Z 333.064,A -85,B 0,C 180,E1 -14531.607,E2 -14531.607} C_VEL
LIN {X 0,Y 351.14,Z 323.564,A -85,B 0,C 180,E1 -14532.857,E2 -14532.857} C_VEL
LIN {X 0,Y 344.378,Z 313.072,A -85,B 0,C 180,E1 -14534.417,E2 -14534.417} C_VEL
LIN {X 0,Y 337.926,Z 303.447,A -85,B 0,C 180,E1 -14536.044,E2 -14536.044} C_VEL
LIN {X 0,Y 333.642,Z 293.222,A -85,B 0,C 180,E1 -14539.233,E2 -14539.233} C_VEL
LIN {X 0,Y 333.664,Z 293.217,A -85,B 0,C 180,E1 -14543.168,E2 -14543.168} C_VEL
LIN {X 0,Y 333.674,Z 293.228,A -85,B 0,C 180,E1 -14545.342,E2 -14545.342} C_VEL
LIN {X 0,Y 333.69,Z 293.231,A -85,B 0,C 180,E1 -14549.638,E2 -14549.638} C_VEL
LIN {X 0,Y 333.74,Z 293.198,A -85,B 0,C 180,E1 -14552.402,E2 -14552.402} C_VEL
LIN {X 0,Y 333.726,Z 293.224,A -85,B 0,C 180,E1 -14555.091,E2 -14555.091} C_VEL
LIN {X 0,Y 333.676,Z 293.22,A -85,B 0,C 180,E1 -14559.02,E2 -14559.02} C_VEL
LIN {X 0,Y 333.795,Z 293.203,A -85,B 0,C 180,E1 -14561.59,E2 -14561.59} C_VEL
LIN {X 0,Y 333.809,Z 293.215,A -85,B 0,C 180,E1 -14565.577,E2 -14565.577} C_VEL
LIN {X 0,Y 333.818,Z 293.181,A -85,B 0,C 180,E1 -14569.078,E2 -14569.078} C_VEL
LIN {X 0,Y 333.959,Z 293.198,A -85,B 0,C 180,E1 -14572.747,E2 -14572.747} C_VEL
LIN {X 0,Y 333.793,Z 293.184,A -85,B 0,C 180,E1 -14575.169,E2 -14575.169} C_VEL
LIN {X 0,Y 334.096,Z 293.168,A -85,B 0,C 180,E1 -14577.589,E2 -14577.589} C_VEL
LIN {X 0,Y 334.172,Z 293.16,A -85,B 0,C 180,E1 -14580.001,E2 -14580.001} C_VEL
LIN {X 0,Y 334.069,Z 293.152,A -85,B 0,C 180,E1 -14582.412,E2 -14582.412} C_VEL
LIN {X 0,Y 333.961,Z 293.18,A -85,B 0,C 180,E1 -14586.534,E2 -14586.534} C_VEL
LIN {X 0,Y 333.823,Z 293.2,A -85,B 0,C 180,E1 -14589.697,E2 -14589.697} C_VEL
LIN {X 0,Y 333.795,Z 293.191,A -85,B 0,C 180,E1 -14593.392,E2 -14593.392} C_VEL
LIN {X 0,Y 333.741,Z 293.221,A -85,B 0,C 180,E1 -14595.889,E2 -14595.889} C_VEL
LIN {X 0,Y 333.655,Z 293.211,A -85,B 0,C 180,E1 -14599.696,E2 -14599.696} C_VEL
LIN {X 0,Y 333.652,Z 293.232,A -85,B 0,C 180,E1 -14602.282,E2 -14602.282} C_VEL
LIN {X 0,Y 333.658,Z 293.222,A -85,B 0,C 180,E1 -14605.078,E2 -14605.078} C_VEL
LIN {X 0,Y 333.63,Z 293.223,A -85,B 0,C 180,E1 -14608.981,E2 -14608.981} C_VEL
LIN {X 0,Y 333.677,Z 293.287,A -85,B 0,C 180,E1 -14610.188,E2 -14610.188} C_VEL
LIN {X 0,Y 334.438,Z 295.72,A -85,B 0,C 180,E1 -14610.438,E2 -14610.438} C_VEL
LIN {X 0,Y 336.223,Z 297.877,A -85,B 0,C 180,E1 -14610.893,E2 -14610.893} C_VEL
LIN {X 0,Y 337.37,Z 298.874,A -85,B 0,C 180,E1 -14611.168,E2 -14611.168} C_VEL
LIN {X 0,Y 339.49,Z 302.208,A -85,B 0,C 180,E1 -14611.716,E2 -14611.716} C_VEL
LIN {X 0,Y 341.09,Z 303.999,A -85,B 0,C 180,E1 -14612.097,E2 -14612.097} C_VEL
LIN {X 0,Y 343.869,Z 307.725,A -85,B 0,C 180,E1 -14612.764,E2 -14612.764} C_VEL
LIN {X 0,Y 351.17,Z 318.008,A -85,B 0,C 180,E1 -14614.429,E2 -14614.429} C_VEL
LIN {X 0,Y 357.148,Z 326.906,A -85,B 0,C 180,E1 -14615.714,E2 -14615.714} C_VEL
LIN {X 0,Y 365.399,Z 341.165,A -85,B 0,C 180,E1 -14617.422,E2 -14617.422} C_VEL
LIN {X 0,Y 370.97,Z 351.595,A -85,B 0,C 180,E1 -14618.523,E2 -14618.523} C_VEL
LIN {X 0,Y 365.089,Z 495.208,A -85,B 0,C 180,E1 -14621.448,E2 -14621.448} C_VEL
LIN {X 0,Y 363.838,Z 511.101,A -85,B 0,C 180,E1 -14621.954,E2 -14621.954} C_VEL
LIN {X 0,Y 362.041,Z 527.112,A -85,B 0,C 180,E1 -14622.662,E2 -14622.662} C_VEL
LIN {X 0,Y 359.862,Z 542.893,A -85,B 0,C 180,E1 -14623.592,E2 -14623.592} C_VEL
LIN {X 0,Y 357.34,Z 558.057,A -85,B 0,C 180,E1 -14624.725,E2 -14624.725} C_VEL
LIN {X 0,Y 354.518,Z 572.523,A -85,B 0,C 180,E1 -14626.065,E2 -14626.065} C_VEL
LIN {X 0,Y 351.524,Z 586.296,A -85,B 0,C 180,E1 -14627.61,E2 -14627.61} C_VEL
LIN {X 0,Y 348.363,Z 599.63,A -85,B 0,C 180,E1 -14629.411,E2 -14629.411} C_VEL
LIN {X 0,Y 345.463,Z 611.224,A -85,B 0,C 180,E1 -14631.276,E2 -14631.276} C_VEL
LIN {X 0,Y 342.394,Z 622.668,A -85,B 0,C 180,E1 -14633.469,E2 -14633.469} C_VEL
LIN {X 0,Y 339.672,Z 632.929,A -85,B 0,C 180,E1 -14635.857,E2 -14635.857} C_VEL
LIN {X 0,Y 337.493,Z 641.537,A -85,B 0,C 180,E1 -14638.277,E2 -14638.277} C_VEL
LIN {X 0,Y 335.779,Z 648.301,A -85,B 0,C 180,E1 -14640.537,E2 -14640.537} C_VEL
LIN {X 0,Y 334.311,Z 654.623,A -85,B 0,C 180,E1 -14643.129,E2 -14643.129} C_VEL
LIN {X 0,Y 333.212,Z 659.616,A -85,B 0,C 180,E1 -14645.714,E2 -14645.714} C_VEL
LIN {X 0,Y 332.505,Z 663.625,A -85,B 0,C 180,E1 -14648.438,E2 -14648.438} C_VEL
LIN {X 0,Y 331.985,Z 666.645,A -85,B 0,C 180,E1 -14651.485,E2 -14651.485} C_VEL
LIN {X 0,Y 331.784,Z 667.977,A -85,B 0,C 180,E1 -14654.016,E2 -14654.016} C_VEL
LIN {X 0,Y 331.845,Z 668.272,A -85,B 0,C 180,E1 -14656.964,E2 -14656.964} C_VEL
LIN {X 0,Y 331.81,Z 667.682,A -85,B 0,C 180,E1 -14659.01,E2 -14659.01} C_VEL
LIN {X 0,Y 331.885,Z 666.061,A -85,B 0,C 180,E1 -14661.475,E2 -14661.475} C_VEL
LIN {X 0,Y 332.204,Z 663.452,A -85,B 0,C 180,E1 -14663.928,E2 -14663.928} C_VEL
LIN {X 0,Y 332.667,Z 658.753,A -85,B 0,C 180,E1 -14666.972,E2 -14666.972} C_VEL
LIN {X 0,Y 333.2,Z 653.801,A -85,B 0,C 180,E1 -14669.396,E2 -14669.396} C_VEL
LIN {X 0,Y 334.221,Z 647.726,A -85,B 0,C 180,E1 -14671.807,E2 -14671.807} C_VEL
LIN {X 0,Y 335.59,Z 639.32,A -85,B 0,C 180,E1 -14674.504,E2 -14674.504} C_VEL
LIN {X 0,Y 337.444,Z 630.265,A -85,B 0,C 180,E1 -14676.878,E2 -14676.878} C_VEL
LIN {X 0,Y 339.611,Z 619.54,A -85,B 0,C 180,E1 -14679.229,E2 -14679.229} C_VEL
LIN {X 0,Y 341.75,Z 608.5,A -85,B 0,C 180,E1 -14681.266,E2 -14681.266} C_VEL
LIN {X 0,Y 344.023,Z 596.523,A -85,B 0,C 180,E1 -14683.136,E2 -14683.136} C_VEL
LIN {X 0,Y 346.396,Z 583.428,A -85,B 0,C 180,E1 -14684.841,E2 -14684.841} C_VEL
LIN {X 0,Y 348.823,Z 569.197,A -85,B 0,C 180,E1 -14686.384,E2 -14686.384} C_VEL
LIN {X 0,Y 351.19,Z 553.592,A -85,B 0,C 180,E1 -14687.769,E2 -14687.769} C_VEL
LIN {X 0,Y 353.111,Z 538.276,A -85,B 0,C 180,E1 -14688.87,E2 -14688.87} C_VEL
LIN {X 0,Y 354.703,Z 523.932,A -85,B 0,C 180,E1 -14689.684,E2 -14689.684} C_VEL
LIN {X 0,Y 355.719,Z 512.222,A -85,B 0,C 180,E1 -14690.208,E2 -14690.208} C_VEL
LIN {X 0,Y 355.666,Z 506.531,A -85,B 0,C 180,E1 -14690.468,E2 -14690.468} C_VEL
LIN {X 0,Y 353.796,Z 497.335,A -85,B 0,C 180,E1 -14690.988,E2 -14690.988} C_VEL
LIN {X 0,Y 351.719,Z 488.077,A -85,B 0,C 180,E1 -14691.457,E2 -14691.457} C_VEL
LIN {X 0,Y 351.33,Z 482.287,A -85,B 0,C 180,E1 -14691.635,E2 -14691.635} C_VEL
LIN {X 0,Y 355.866,Z 348.812,A -85,B 0,C 180,E1 -14694.341,E2 -14694.341} C_VEL
LIN {X 0,Y 354.176,Z 344.47,A -85,B 0,C 180,E1 -14694.627,E2 -14694.627} C_VEL
LIN {X 0,Y 343.97,Z 323.717,A -85,B 0,C 180,E1 -14696.289,E2 -14696.289} C_VEL
LIN {X 0,Y 333.134,Z 305.498,A -85,B 0,C 180,E1 -14698.101,E2 -14698.101} C_VEL
LIN {X 0,Y 329.1,Z 298.927,A -85,B 0,C 180,E1 -14698.807,E2 -14698.807} C_VEL
LIN {X 0,Y 327.051,Z 295.862,A -85,B 0,C 180,E1 -14699.168,E2 -14699.168} C_VEL
LIN {X 0,Y 326.585,Z 294.116,A -85,B 0,C 180,E1 -14699.299,E2 -14699.299} C_VEL
LIN {X 0,Y 326.617,Z 294.113,A -85,B 0,C 180,E1 -14702.945,E2 -14702.945} C_VEL
LIN {X 0,Y 326.613,Z 294.106,A -85,B 0,C 180,E1 -14705.52,E2 -14705.52} C_VEL
LIN {X 0,Y 326.573,Z 294.114,A -85,B 0,C 180,E1 -14709.218,E2 -14709.218} C_VEL
LIN {X 0,Y 326.574,Z 294.111,A -85,B 0,C 180,E1 -14712.97,E2 -14712.97} C_VEL
LIN {X 0,Y 326.573,Z 294.105,A -85,B 0,C 180,E1 -14717.029,E2 -14717.029} C_VEL
LIN {X 0,Y 326.588,Z 294.099,A -85,B 0,C 180,E1 -14720.778,E2 -14720.778} C_VEL
LIN {X 0,Y 326.611,Z 294.066,A -85,B 0,C 180,E1 -14724.479,E2 -14724.479} C_VEL
LIN {X 0,Y 326.61,Z 294.11,A -85,B 0,C 180,E1 -14727.455,E2 -14727.455} C_VEL
LIN {X 0,Y 326.582,Z 294.101,A -85,B 0,C 180,E1 -14730.332,E2 -14730.332} C_VEL
LIN {X 0,Y 326.609,Z 294.112,A -85,B 0,C 180,E1 -14733.135,E2 -14733.135} C_VEL
LIN {X 0,Y 326.63,Z 294.095,A -85,B 0,C 180,E1 -14735.869,E2 -14735.869} C_VEL
LIN {X 0,Y 326.633,Z 294.109,A -85,B 0,C 180,E1 -14739.862,E2 -14739.862} C_VEL
LIN {X 0,Y 326.665,Z 294.09,A -85,B 0,C 180,E1 -14742.469,E2 -14742.469} C_VEL
LIN {X 0,Y 326.76,Z 294.09,A -85,B 0,C 180,E1 -14746.314,E2 -14746.314} C_VEL
LIN {X 0,Y 326.805,Z 294.088,A -85,B 0,C 180,E1 -14750.093,E2 -14750.093} C_VEL
LIN {X 0,Y 326.963,Z 294.051,A -85,B 0,C 180,E1 -14753.83,E2 -14753.83} C_VEL
LIN {X 0,Y 327.034,Z 294.062,A -85,B 0,C 180,E1 -14757.536,E2 -14757.536} C_VEL
LIN {X 0,Y 327.178,Z 294.023,A -85,B 0,C 180,E1 -14759.999,E2 -14759.999} C_VEL
LIN {X 0,Y 327.046,Z 294.056,A -85,B 0,C 180,E1 -14762.463,E2 -14762.463} C_VEL
LIN {X 0,Y 326.963,Z 294.048,A -85,B 0,C 180,E1 -14766.169,E2 -14766.169} C_VEL
LIN {X 0,Y 326.911,Z 294.063,A -85,B 0,C 180,E1 -14768.655,E2 -14768.655} C_VEL
LIN {X 0,Y 326.734,Z 294.092,A -85,B 0,C 180,E1 -14772.421,E2 -14772.421} C_VEL
LIN {X 0,Y 326.75,Z 294.097,A -85,B 0,C 180,E1 -14774.957,E2 -14774.957} C_VEL
LIN {X 0,Y 326.706,Z 294.1,A -85,B 0,C 180,E1 -14778.824,E2 -14778.824} C_VEL
LIN {X 0,Y 326.62,Z 294.11,A -85,B 0,C 180,E1 -14782.787,E2 -14782.787} C_VEL
LIN {X 0,Y 326.689,Z 294.103,A -85,B 0,C 180,E1 -14785.483,E2 -14785.483} C_VEL
LIN {X 0,Y 326.646,Z 294.11,A -85,B 0,C 180,E1 -14789.66,E2 -14789.66} C_VEL
LIN {X 0,Y 326.605,Z 294.114,A -85,B 0,C 180,E1 -14794.019,E2 -14794.019} C_VEL
LIN {X 0,Y 326.626,Z 294.098,A -85,B 0,C 180,E1 -14797.238,E2 -14797.238} C_VEL
LIN {X 0,Y 326.575,Z 294.107,A -85,B 0,C 180,E1 -14801.131,E2 -14801.131} C_VEL
LIN {X 0,Y 326.557,Z 294.112,A -85,B 0,C 180,E1 -14804.748,E2 -14804.748} C_VEL
LIN {X 0,Y 326.602,Z 294.146,A -85,B 0,C 180,E1 -14805.741,E2 -14805.741} C_VEL
LIN {X 0,Y 330.495,Z 305.084,A -85,B 0,C 180,E1 -14808.158,E2 -14808.158} C_VEL
LIN {X 0,Y 338.646,Z 320.144,A -85,B 0,C 180,E1 -14809.594,E2 -14809.594} C_VEL
LIN {X 0,Y 347.918,Z 338.774,A -85,B 0,C 180,E1 -14811.158,E2 -14811.158} C_VEL
LIN {X 0,Y 355.749,Z 356.053,A -85,B 0,C 180,E1 -14812.436,E2 -14812.436} C_VEL
LIN {X 0,Y 350.518,Z 512.167,A -85,B 0,C 180,E1 -14815.638,E2 -14815.638} C_VEL
LIN {X 0,Y 349.345,Z 528.196,A -85,B 0,C 180,E1 -14816.151,E2 -14816.151} C_VEL
LIN {X 0,Y 347.616,Z 545.08,A -85,B 0,C 180,E1 -14816.915,E2 -14816.915} C_VEL
LIN {X 0,Y 345.777,Z 560.391,A -85,B 0,C 180,E1 -14817.841,E2 -14817.841} C_VEL
LIN {X 0,Y 343.55,Z 574.592,A -85,B 0,C 180,E1 -14818.9,E2 -14818.9} C_VEL
LIN {X 0,Y 341.342,Z 588.404,A -85,B 0,C 180,E1 -14820.182,E2 -14820.182} C_VEL
LIN {X 0,Y 338.872,Z 601.958,A -85,B 0,C 180,E1 -14821.679,E2 -14821.679} C_VEL
LIN {X 0,Y 336.278,Z 615.45,A -85,B 0,C 180,E1 -14823.466,E2 -14823.466} C_VEL
LIN {X 0,Y 333.821,Z 627.815,A -85,B 0,C 180,E1 -14825.43,E2 -14825.43} C_VEL
LIN {X 0,Y 331.501,Z 639.097,A -85,B 0,C 180,E1 -14827.567,E2 -14827.567} C_VEL
LIN {X 0,Y 329.595,Z 648.855,A -85,B 0,C 180,E1 -14829.753,E2 -14829.753} C_VEL
LIN {X 0,Y 327.958,Z 658.125,A -85,B 0,C 180,E1 -14832.22,E2 -14832.22} C_VEL
LIN {X 0,Y 326.553,Z 666.791,A -85,B 0,C 180,E1 -14835.033,E2 -14835.033} C_VEL
LIN {X 0,Y 325.693,Z 673.017,A -85,B 0,C 180,E1 -14837.538,E2 -14837.538} C_VEL
LIN {X 0,Y 325.154,Z 678.041,A -85,B 0,C 180,E1 -14840.043,E2 -14840.043} C_VEL
LIN {X 0,Y 324.942,Z 681.977,A -85,B 0,C 180,E1 -14842.544,E2 -14842.544} C_VEL
LIN {X 0,Y 324.86,Z 684.776,A -85,B 0,C 180,E1 -14845.036,E2 -14845.036} C_VEL
LIN {X 0,Y 324.833,Z 686.629,A -85,B 0,C 180,E1 -14847.52,E2 -14847.52} C_VEL
LIN {X 0,Y 324.872,Z 687.408,A -85,B 0,C 180,E1 -14850,E2 -14850} C_VEL
LIN {X 0,Y 324.826,Z 687.294,A -85,B 0,C 180,E1 -14852.48,E2 -14852.48} C_VEL
LIN {X 0,Y 324.844,Z 686.135,A -85,B 0,C 180,E1 -14854.965,E2 -14854.965} C_VEL
LIN {X 0,Y 324.943,Z 684.084,A -85,B 0,C 180,E1 -14857.456,E2 -14857.456} C_VEL
LIN {X 0,Y 325.201,Z 680.962,A -85,B 0,C 180,E1 -14859.956,E2 -14859.956} C_VEL
LIN {X 0,Y 325.85,Z 676.901,A -85,B 0,C 180,E1 -14862.456,E2 -14862.456} C_VEL
LIN {X 0,Y 327.02,Z 670.223,A -85,B 0,C 180,E1 -14865.583,E2 -14865.583} C_VEL
LIN {X 0,Y 329.055,Z 661.68,A -85,B 0,C 180,E1 -14868.686,E2 -14868.686} C_VEL
LIN {X 0,Y 331.385,Z 652.158,A -85,B 0,C 180,E1 -14871.459,E2 -14871.459} C_VEL
LIN {X 0,Y 334.125,Z 641.971,A -85,B 0,C 180,E1 -14873.885,E2 -14873.885} C_VEL
LIN {X 0,Y 336.911,Z 631.516,A -85,B 0,C 180,E1 -14875.98,E2 -14875.98} C_VEL
LIN {X 0,Y 339.636,Z 621.233,A -85,B 0,C 180,E1 -14877.748,E2 -14877.748} C_VEL
LIN {X 0,Y 343.231,Z 607.089,A -85,B 0,C 180,E1 -14879.772,E2 -14879.772} C_VEL
LIN {X 0,Y 346.325,Z 594.04,A -85,B 0,C 180,E1 -14881.307,E2 -14881.307} C_VEL
LIN {X 0,Y 349.477,Z 579.612,A -85,B 0,C 180,E1 -14882.715,E2 -14882.715} C_VEL
LIN {X 0,Y 352.511,Z 564.149,A -85,B 0,C 180,E1 -14883.934,E2 -14883.934} C_VEL
LIN {X 0,Y 354.931,Z 549.402,A -85,B 0,C 180,E1 -14884.873,E2 -14884.873} C_VEL
LIN {X 0,Y 357.001,Z 533.77,A -85,B 0,C 180,E1 -14885.633,E2 -14885.633} C_VEL
LIN {X 0,Y 358.696,Z 517.261,A -85,B 0,C 180,E1 -14886.213,E2 -14886.213} C_VEL
LIN {X 0,Y 359.861,Z 497.602,A -85,B 0,C 180,E1 -14886.673,E2 -14886.673} C_VEL
LIN {X 0,Y 365.411,Z 361.851,A -85,B 0,C 180,E1 -14889.466,E2 -14889.466} C_VEL
LIN {X 0,Y 358.622,Z 348.277,A -85,B 0,C 180,E1 -14890.886,E2 -14890.886} C_VEL
LIN {X 0,Y 350.578,Z 333.894,A -85,B 0,C 180,E1 -14892.648,E2 -14892.648} C_VEL
LIN {X 0,Y 341.662,Z 319.591,A -85,B 0,C 180,E1 -14894.734,E2 -14894.734} C_VEL
LIN {X 0,Y 333.848,Z 308.151,A -85,B 0,C 180,E1 -14896.712,E2 -14896.712} C_VEL
LIN {X 0,Y 330.303,Z 303.026,A -85,B 0,C 180,E1 -14897.71,E2 -14897.71} C_VEL
LIN {X 0,Y 326.605,Z 294.115,A -85,B 0,C 180,E1 -14900.69,E2 -14900.69} C_VEL
LIN {X 0,Y 326.613,Z 294.113,A -85,B 0,C 180,E1 -14904.481,E2 -14904.481} C_VEL
LIN {X 0,Y 326.607,Z 294.091,A -85,B 0,C 180,E1 -14907.456,E2 -14907.456} C_VEL
LIN {X 0,Y 326.648,Z 294.096,A -85,B 0,C 180,E1 -14910.34,E2 -14910.34} C_VEL
LIN {X 0,Y 326.69,Z 294.104,A -85,B 0,C 180,E1 -14914.517,E2 -14914.517} C_VEL
LIN {X 0,Y 326.621,Z 294.09,A -85,B 0,C 180,E1 -14918.544,E2 -14918.544} C_VEL
LIN {X 0,Y 326.745,Z 294.089,A -85,B 0,C 180,E1 -14921.178,E2 -14921.178} C_VEL
LIN {X 0,Y 326.764,Z 294.089,A -85,B 0,C 180,E1 -14925.434,E2 -14925.434} C_VEL
LIN {X 0,Y 326.759,Z 294.061,A -85,B 0,C 180,E1 -14928.839,E2 -14928.839} C_VEL
LIN {X 0,Y 326.915,Z 294.077,A -85,B 0,C 180,E1 -14932.59,E2 -14932.59} C_VEL
LIN {X 0,Y 326.761,Z 294.06,A -85,B 0,C 180,E1 -14935.065,E2 -14935.065} C_VEL
LIN {X 0,Y 327.036,Z 294.045,A -85,B 0,C 180,E1 -14937.537,E2 -14937.537} C_VEL
LIN {X 0,Y 327.127,Z 294.037,A -85,B 0,C 180,E1 -14940.001,E2 -14940.001} C_VEL
LIN {X 0,Y 327.012,Z 294.03,A -85,B 0,C 180,E1 -14942.464,E2 -14942.464} C_VEL
LIN {X 0,Y 326.922,Z 294.057,A -85,B 0,C 180,E1 -14946.524,E2 -14946.524} C_VEL
LIN {X 0,Y 326.785,Z 294.08,A -85,B 0,C 180,E1 -14949.908,E2 -14949.908} C_VEL
LIN {X 0,Y 326.759,Z 294.066,A -85,B 0,C 180,E1 -14953.686,E2 -14953.686} C_VEL
LIN {X 0,Y 326.637,Z 294.099,A -85,B 0,C 180,E1 -14957.532,E2 -14957.532} C_VEL
LIN {X 0,Y 326.61,Z 294.092,A -85,B 0,C 180,E1 -14960.139,E2 -14960.139} C_VEL
LIN {X 0,Y 326.593,Z 294.101,A -85,B 0,C 180,E1 -14962.79,E2 -14962.79} C_VEL
LIN {X 0,Y 326.597,Z 294.107,A -85,B 0,C 180,E1 -14966.866,E2 -14966.866} C_VEL
LIN {X 0,Y 326.596,Z 294.2,A -85,B 0,C 180,E1 -14968.608,E2 -14968.608} C_VEL
LIN {X 0,Y 327.498,Z 296.805,A -85,B 0,C 180,E1 -14968.916,E2 -14968.916} C_VEL
LIN {X 0,Y 329.497,Z 298.975,A -85,B 0,C 180,E1 -14969.454,E2 -14969.454} C_VEL
LIN {X 0,Y 330.446,Z 299.802,A -85,B 0,C 180,E1 -14969.698,E2 -14969.698} C_VEL
LIN {X 0,Y 332.369,Z 302.92,A -85,B 0,C 180,E1 -14970.235,E2 -14970.235} C_VEL
LIN {X 0,Y 334.36,Z 305.14,A -85,B 0,C 180,E1 -14970.743,E2 -14970.743} C_VEL
LIN {X 0,Y 337.145,Z 308.82,A -85,B 0,C 180,E1 -14971.453,E2 -14971.453} C_VEL
LIN {X 0,Y 344.568,Z 319.044,A -85,B 0,C 180,E1 -14973.252,E2 -14973.252} C_VEL
LIN {X 0,Y 352.577,Z 330.776,A -85,B 0,C 180,E1 -14975.053,E2 -14975.053} C_VEL
LIN {X 0,Y 361.138,Z 345.688,A -85,B 0,C 180,E1 -14976.888,E2 -14976.888} C_VEL
LIN {X 0,Y 365.616,Z 354.118,A -85,B 0,C 180,E1 -14977.804,E2 -14977.804} C_VEL
LIN {X 0,Y 362.401,Z 431.431,A -85,B 0,C 180,E1 -14979.393,E2 -14979.393} C_VEL
LIN {X 0,Y 359.668,Z 495.487,A -85,B 0,C 180,E1 -14980.73,E2 -14980.73} C_VEL
LIN {X 0,Y 358.361,Z 511.323,A -85,B 0,C 180,E1 -14981.238,E2 -14981.238} C_VEL
LIN {X 0,Y 356.628,Z 526.492,A -85,B 0,C 180,E1 -14981.911,E2 -14981.911} C_VEL
LIN {X 0,Y 354.468,Z 541.889,A -85,B 0,C 180,E1 -14982.811,E2 -14982.811} C_VEL
LIN {X 0,Y 352.052,Z 555.909,A -85,B 0,C 180,E1 -14983.849,E2 -14983.849} C_VEL
LIN {X 0,Y 349.068,Z 570.816,A -85,B 0,C 180,E1 -14985.196,E2 -14985.196} C_VEL
LIN {X 0,Y 346.14,Z 583.96,A -85,B 0,C 180,E1 -14986.636,E2 -14986.636} C_VEL
LIN {X 0,Y 342.89,Z 597.506,A -85,B 0,C 180,E1 -14988.427,E2 -14988.427} C_VEL
LIN {X 0,Y 340.029,Z 608.417,A -85,B 0,C 180,E1 -14990.153,E2 -14990.153} C_VEL
LIN {X 0,Y 336.727,Z 620.27,A -85,B 0,C 180,E1 -14992.366,E2 -14992.366} C_VEL
LIN {X 0,Y 333.891,Z 630.361,A -85,B 0,C 180,E1 -14994.631,E2 -14994.631} C_VEL
LIN {X 0,Y 331.584,Z 638.921,A -85,B 0,C 180,E1 -14996.922,E2 -14996.922} C_VEL
LIN {X 0,Y 329.608,Z 646.063,A -85,B 0,C 180,E1 -14999.22,E2 -14999.22} C_VEL
LIN {X 0,Y 327.923,Z 652.874,A -85,B 0,C 180,E1 -15001.868,E2 -15001.868} C_VEL
LIN {X 0,Y 326.545,Z 658.653,A -85,B 0,C 180,E1 -15004.682,E2 -15004.682} C_VEL
LIN {X 0,Y 325.736,Z 662.501,A -85,B 0,C 180,E1 -15007.147,E2 -15007.147} C_VEL
LIN {X 0,Y 325.124,Z 665.568,A -85,B 0,C 180,E1 -15009.765,E2 -15009.765} C_VEL
LIN {X 0,Y 324.862,Z 667.526,A -85,B 0,C 180,E1 -15012.37,E2 -15012.37} C_VEL
LIN {X 0,Y 324.662,Z 668.455,A -85,B 0,C 180,E1 -15014.944,E2 -15014.944} C_VEL
LIN {X 0,Y 324.744,Z 668.396,A -85,B 0,C 180,E1 -15017.501,E2 -15017.501} C_VEL
LIN {X 0,Y 324.681,Z 667.326,A -85,B 0,C 180,E1 -15020.028,E2 -15020.028} C_VEL
LIN {X 0,Y 324.9,Z 665.321,A -85,B 0,C 180,E1 -15022.543,E2 -15022.543} C_VEL
LIN {X 0,Y 325.222,Z 662.255,A -85,B 0,C 180,E1 -15025.041,E2 -15025.041} C_VEL
LIN {X 0,Y 325.702,Z 658.242,A -85,B 0,C 180,E1 -15027.526,E2 -15027.526} C_VEL
LIN {X 0,Y 326.571,Z 651.645,A -85,B 0,C 180,E1 -15030.616,E2 -15030.616} C_VEL
LIN {X 0,Y 327.674,Z 644.978,A -85,B 0,C 180,E1 -15033.074,E2 -15033.074} C_VEL
LIN {X 0,Y 329.168,Z 637.017,A -85,B 0,C 180,E1 -15035.513,E2 -15035.513} C_VEL
LIN {X 0,Y 331.208,Z 627.538,A -85,B 0,C 180,E1 -15037.928,E2 -15037.928} C_VEL
LIN {X 0,Y 333.263,Z 617.766,A -85,B 0,C 180,E1 -15040.019,E2 -15040.019} C_VEL
LIN {X 0,Y 335.58,Z 606.326,A -85,B 0,C 180,E1 -15042.089,E2 -15042.089} C_VEL
LIN {X 0,Y 337.988,Z 593.889,A -85,B 0,C 180,E1 -15043.988,E2 -15043.988} C_VEL
LIN {X 0,Y 340.461,Z 580.37,A -85,B 0,C 180,E1 -15045.72,E2 -15045.72} C_VEL
LIN {X 0,Y 342.855,Z 566.992,A -85,B 0,C 180,E1 -15047.137,E2 -15047.137} C_VEL
LIN {X 0,Y 345.068,Z 552.549,A -85,B 0,C 180,E1 -15048.402,E2 -15048.402} C_VEL
LIN {X 0,Y 346.975,Z 536.928,A -85,B 0,C 180,E1 -15049.524,E2 -15049.524} C_VEL
LIN {X 0,Y 348.84,Z 520.629,A -85,B 0,C 180,E1 -15050.413,E2 -15050.413} C_VEL
LIN {X 0,Y 350.175,Z 504.787,A -85,B 0,C 180,E1 -15051.062,E2 -15051.062} C_VEL
LIN {X 0,Y 351.12,Z 488.505,A -85,B 0,C 180,E1 -15051.502,E2 -15051.502} C_VEL
LIN {X 0,Y 351.33,Z 482.287,A -85,B 0,C 180,E1 -15051.635,E2 -15051.635} C_VEL
LIN {X 0,Y 350.945,Z 476.487,A -85,B 0,C 180,E1 -15051.809,E2 -15051.809} C_VEL
LIN {X 0,Y 346.635,Z 457.864,A -85,B 0,C 180,E1 -15052.685,E2 -15052.685} C_VEL
LIN {X 0,Y 346.301,Z 452.063,A -85,B 0,C 180,E1 -15052.86,E2 -15052.86} C_VEL
LIN {X 0,Y 349.902,Z 350.476,A -85,B 0,C 180,E1 -15054.948,E2 -15054.948} C_VEL
LIN {X 0,Y 339.938,Z 329.559,A -85,B 0,C 180,E1 -15056.621,E2 -15056.621} C_VEL
LIN {X 0,Y 328.594,Z 310.26,A -85,B 0,C 180,E1 -15058.567,E2 -15058.567} C_VEL
LIN {X 0,Y 322.22,Z 300.033,A -85,B 0,C 180,E1 -15059.722,E2 -15059.722} C_VEL
LIN {X 0,Y 320.009,Z 296.791,A -85,B 0,C 180,E1 -15060.129,E2 -15060.129} C_VEL
LIN {X 0,Y 319.568,Z 294.993,A -85,B 0,C 180,E1 -15060.279,E2 -15060.279} C_VEL
LIN {X 0,Y 319.579,Z 294.991,A -85,B 0,C 180,E1 -15063.352,E2 -15063.352} C_VEL
LIN {X 0,Y 319.557,Z 294.994,A -85,B 0,C 180,E1 -15066.428,E2 -15066.428} C_VEL
LIN {X 0,Y 319.531,Z 294.994,A -85,B 0,C 180,E1 -15069.661,E2 -15069.661} C_VEL
LIN {X 0,Y 319.52,Z 294.993,A -85,B 0,C 180,E1 -15073.459,E2 -15073.459} C_VEL
LIN {X 0,Y 319.552,Z 294.979,A -85,B 0,C 180,E1 -15077.015,E2 -15077.015} C_VEL
LIN {X 0,Y 319.547,Z 294.983,A -85,B 0,C 180,E1 -15080.37,E2 -15080.37} C_VEL
LIN {X 0,Y 319.579,Z 294.94,A -85,B 0,C 180,E1 -15084.457,E2 -15084.457} C_VEL
LIN {X 0,Y 319.526,Z 294.997,A -85,B 0,C 180,E1 -15088.137,E2 -15088.137} C_VEL
LIN {X 0,Y 319.546,Z 294.979,A -85,B 0,C 180,E1 -15091.612,E2 -15091.612} C_VEL
LIN {X 0,Y 319.572,Z 294.979,A -85,B 0,C 180,E1 -15095.301,E2 -15095.301} C_VEL
LIN {X 0,Y 319.567,Z 294.987,A -85,B 0,C 180,E1 -15098.045,E2 -15098.045} C_VEL
LIN {X 0,Y 319.626,Z 294.965,A -85,B 0,C 180,E1 -15102.07,E2 -15102.07} C_VEL
LIN {X 0,Y 319.733,Z 294.966,A -85,B 0,C 180,E1 -15106.007,E2 -15106.007} C_VEL
LIN {X 0,Y 319.752,Z 294.962,A -85,B 0,C 180,E1 -15109.872,E2 -15109.872} C_VEL
LIN {X 0,Y 319.92,Z 294.929,A -85,B 0,C 180,E1 -15113.693,E2 -15113.693} C_VEL
LIN {X 0,Y 319.978,Z 294.941,A -85,B 0,C 180,E1 -15117.482,E2 -15117.482} C_VEL
LIN {X 0,Y 320.13,Z 294.9,A -85,B 0,C 180,E1 -15119.999,E2 -15119.999} C_VEL
LIN {X 0,Y 319.989,Z 294.935,A -85,B 0,C 180,E1 -15122.517,E2 -15122.517} C_VEL
LIN {X 0,Y 319.922,Z 294.923,A -85,B 0,C 180,E1 -15126.305,E2 -15126.305} C_VEL
LIN {X 0,Y 319.838,Z 294.945,A -85,B 0,C 180,E1 -15128.847,E2 -15128.847} C_VEL
LIN {X 0,Y 319.681,Z 294.971,A -85,B 0,C 180,E1 -15132.699,E2 -15132.699} C_VEL
LIN {X 0,Y 319.678,Z 294.974,A -85,B 0,C 180,E1 -15135.296,E2 -15135.296} C_VEL
LIN {X 0,Y 319.653,Z 294.978,A -85,B 0,C 180,E1 -15139.256,E2 -15139.256} C_VEL
LIN {X 0,Y 319.569,Z 294.994,A -85,B 0,C 180,E1 -15143.319,E2 -15143.319} C_VEL
LIN {X 0,Y 319.633,Z 294.984,A -85,B 0,C 180,E1 -15146.088,E2 -15146.088} C_VEL
LIN {X 0,Y 319.579,Z 294.99,A -85,B 0,C 180,E1 -15148.934,E2 -15148.934} C_VEL
LIN {X 0,Y 319.529,Z 294.997,A -85,B 0,C 180,E1 -15151.861,E2 -15151.861} C_VEL
LIN {X 0,Y 319.578,Z 294.982,A -85,B 0,C 180,E1 -15155.543,E2 -15155.543} C_VEL
LIN {X 0,Y 319.571,Z 294.985,A -85,B 0,C 180,E1 -15158.007,E2 -15158.007} C_VEL
LIN {X 0,Y 319.523,Z 294.988,A -85,B 0,C 180,E1 -15161.597,E2 -15161.597} C_VEL
LIN {X 0,Y 319.523,Z 295.056,A -85,B 0,C 180,E1 -15164.895,E2 -15164.895} C_VEL
LIN {X 0,Y 323.075,Z 304.751,A -85,B 0,C 180,E1 -15167.144,E2 -15167.144} C_VEL
LIN {X 0,Y 332.868,Z 322.616,A -85,B 0,C 180,E1 -15168.936,E2 -15168.936} C_VEL
LIN {X 0,Y 342.543,Z 342.121,A -85,B 0,C 180,E1 -15170.623,E2 -15170.623} C_VEL
LIN {X 0,Y 349.722,Z 358.135,A -85,B 0,C 180,E1 -15171.836,E2 -15171.836} C_VEL
LIN {X 0,Y 345.566,Z 479.336,A -85,B 0,C 180,E1 -15174.339,E2 -15174.339} C_VEL
LIN {X 0,Y 344.289,Z 514.275,A -85,B 0,C 180,E1 -15175.105,E2 -15175.105} C_VEL
LIN {X 0,Y 342.885,Z 531.433,A -85,B 0,C 180,E1 -15175.691,E2 -15175.691} C_VEL
LIN {X 0,Y 341.126,Z 547.345,A -85,B 0,C 180,E1 -15176.468,E2 -15176.468} C_VEL
LIN {X 0,Y 339.065,Z 563.09,A -85,B 0,C 180,E1 -15177.478,E2 -15177.478} C_VEL
LIN {X 0,Y 336.701,Z 577.877,A -85,B 0,C 180,E1 -15178.657,E2 -15178.657} C_VEL
LIN {X 0,Y 334.273,Z 592.039,A -85,B 0,C 180,E1 -15180.044,E2 -15180.044} C_VEL
LIN {X 0,Y 331.801,Z 604.691,A -85,B 0,C 180,E1 -15181.538,E2 -15181.538} C_VEL
LIN {X 0,Y 329.143,Z 617.685,A -85,B 0,C 180,E1 -15183.359,E2 -15183.359} C_VEL
LIN {X 0,Y 326.875,Z 628.875,A -85,B 0,C 180,E1 -15185.212,E2 -15185.212} C_VEL
LIN {X 0,Y 324.499,Z 639.995,A -85,B 0,C 180,E1 -15187.392,E2 -15187.392} C_VEL
LIN {X 0,Y 322.381,Z 650.726,A -85,B 0,C 180,E1 -15189.919,E2 -15189.919} C_VEL
LIN {X 0,Y 320.652,Z 659.696,A -85,B 0,C 180,E1 -15192.46,E2 -15192.46} C_VEL
LIN {X 0,Y 319.335,Z 667.885,A -85,B 0,C 180,E1 -15195.289,E2 -15195.289} C_VEL
LIN {X 0,Y 318.506,Z 674.029,A -85,B 0,C 180,E1 -15197.9,E2 -15197.9} C_VEL
LIN {X 0,Y 318.014,Z 678.783,A -85,B 0,C 180,E1 -15200.459,E2 -15200.459} C_VEL
LIN {X 0,Y 317.857,Z 681.657,A -85,B 0,C 180,E1 -15202.377,E2 -15202.377} C_VEL
LIN {X 0,Y 317.776,Z 684.499,A -85,B 0,C 180,E1 -15204.925,E2 -15204.925} C_VEL
LIN {X 0,Y 317.754,Z 686.372,A -85,B 0,C 180,E1 -15207.465,E2 -15207.465} C_VEL
LIN {X 0,Y 317.78,Z 687.19,A -85,B 0,C 180,E1 -15210,E2 -15210} C_VEL
LIN {X 0,Y 317.746,Z 687.096,A -85,B 0,C 180,E1 -15212.536,E2 -15212.536} C_VEL
LIN {X 0,Y 317.803,Z 685.602,A -85,B 0,C 180,E1 -15215.655,E2 -15215.655} C_VEL
LIN {X 0,Y 317.859,Z 683.947,A -85,B 0,C 180,E1 -15217.624,E2 -15217.624} C_VEL
LIN {X 0,Y 318.134,Z 680.87,A -85,B 0,C 180,E1 -15220.18,E2 -15220.18} C_VEL
LIN {X 0,Y 318.83,Z 676.835,A -85,B 0,C 180,E1 -15222.735,E2 -15222.735} C_VEL
LIN {X 0,Y 319.783,Z 671.633,A -85,B 0,C 180,E1 -15225.292,E2 -15225.292} C_VEL
LIN {X 0,Y 321.292,Z 665.34,A -85,B 0,C 180,E1 -15227.833,E2 -15227.833} C_VEL
LIN {X 0,Y 323.261,Z 657.716,A -85,B 0,C 180,E1 -15230.356,E2 -15230.356} C_VEL
LIN {X 0,Y 325.707,Z 648.636,A -85,B 0,C 180,E1 -15232.855,E2 -15232.855} C_VEL
LIN {X 0,Y 328.755,Z 637.884,A -85,B 0,C 180,E1 -15235.312,E2 -15235.312} C_VEL
LIN {X 0,Y 331.924,Z 626.634,A -85,B 0,C 180,E1 -15237.46,E2 -15237.46} C_VEL
LIN {X 0,Y 335.395,Z 613.831,A -85,B 0,C 180,E1 -15239.501,E2 -15239.501} C_VEL
LIN {X 0,Y 338.911,Z 600.586,A -85,B 0,C 180,E1 -15241.227,E2 -15241.227} C_VEL
LIN {X 0,Y 341.863,Z 587.916,A -85,B 0,C 180,E1 -15242.624,E2 -15242.624} C_VEL
LIN {X 0,Y 344.952,Z 573.949,A -85,B 0,C 180,E1 -15243.899,E2 -15243.899} C_VEL
LIN {X 0,Y 347.903,Z 558.243,A -85,B 0,C 180,E1 -15245.063,E2 -15245.063} C_VEL
LIN {X 0,Y 350.459,Z 541.803,A -85,B 0,C 180,E1 -15246.003,E2 -15246.003} C_VEL
LIN {X 0,Y 352.504,Z 525.421,A -85,B 0,C 180,E1 -15246.691,E2 -15246.691} C_VEL
LIN {X 0,Y 353.979,Z 508.618,A -85,B 0,C 180,E1 -15247.178,E2 -15247.178} C_VEL
LIN {X 0,Y 360.204,Z 365.23,A -85,B 0,C 180,E1 -15250.165,E2 -15250.165} C_VEL
LIN {X 0,Y 359.782,Z 363.529,A -85,B 0,C 180,E1 -15250.278,E2 -15250.278} C_VEL
LIN {X 0,Y 352.632,Z 349.517,A -85,B 0,C 180,E1 -15251.837,E2 -15251.837} C_VEL
LIN {X 0,Y 344.44,Z 334.999,A -85,B 0,C 180,E1 -15253.723,E2 -15253.723} C_VEL
LIN {X 0,Y 336.672,Z 322.761,A -85,B 0,C 180,E1 -15255.629,E2 -15255.629} C_VEL
LIN {X 0,Y 330.445,Z 313.523,A -85,B 0,C 180,E1 -15257.267,E2 -15257.267} C_VEL
LIN {X 0,Y 325.108,Z 306.2,A -85,B 0,C 180,E1 -15258.752,E2 -15258.752} C_VEL
LIN {X 0,Y 322.852,Z 302.676,A -85,B 0,C 180,E1 -15259.475,E2 -15259.475} C_VEL
LIN {X 0,Y 319.55,Z 294.972,A -85,B 0,C 180,E1 -15262.286,E2 -15262.286} C_VEL
LIN {X 0,Y 319.56,Z 294.989,A -85,B 0,C 180,E1 -15265.124,E2 -15265.124} C_VEL
LIN {X 0,Y 319.566,Z 294.989,A -85,B 0,C 180,E1 -15269.06,E2 -15269.06} C_VEL
LIN {X 0,Y 319.605,Z 294.958,A -85,B 0,C 180,E1 -15272.499,E2 -15272.499} C_VEL
LIN {X 0,Y 319.604,Z 294.98,A -85,B 0,C 180,E1 -15275.305,E2 -15275.305} C_VEL
LIN {X 0,Y 319.604,Z 294.979,A -85,B 0,C 180,E1 -15279.401,E2 -15279.401} C_VEL
LIN {X 0,Y 319.659,Z 294.953,A -85,B 0,C 180,E1 -15282.074,E2 -15282.074} C_VEL
LIN {X 0,Y 319.733,Z 294.97,A -85,B 0,C 180,E1 -15286.009,E2 -15286.009} C_VEL
LIN {X 0,Y 319.736,Z 294.935,A -85,B 0,C 180,E1 -15289.873,E2 -15289.873} C_VEL
LIN {X 0,Y 319.903,Z 294.935,A -85,B 0,C 180,E1 -15293.694,E2 -15293.694} C_VEL
LIN {X 0,Y 319.98,Z 294.922,A -85,B 0,C 180,E1 -15297.483,E2 -15297.483} C_VEL
LIN {X 0,Y 320.083,Z 294.914,A -85,B 0,C 180,E1 -15300.001,E2 -15300.001} C_VEL
LIN {X 0,Y 319.958,Z 294.908,A -85,B 0,C 180,E1 -15302.519,E2 -15302.519} C_VEL
LIN {X 0,Y 319.885,Z 294.934,A -85,B 0,C 180,E1 -15306.506,E2 -15306.506} C_VEL
LIN {X 0,Y 319.738,Z 294.961,A -85,B 0,C 180,E1 -15310.128,E2 -15310.128} C_VEL
LIN {X 0,Y 319.732,Z 294.94,A -85,B 0,C 180,E1 -15313.993,E2 -15313.993} C_VEL
LIN {X 0,Y 319.591,Z 294.969,A -85,B 0,C 180,E1 -15317.932,E2 -15317.932} C_VEL
LIN {X 0,Y 319.565,Z 294.99,A -85,B 0,C 180,E1 -15321.955,E2 -15321.955} C_VEL
LIN {X 0,Y 319.551,Z 294.995,A -85,B 0,C 180,E1 -15326.096,E2 -15326.096} C_VEL
LIN {X 0,Y 319.567,Z 295.079,A -85,B 0,C 180,E1 -15326.887,E2 -15326.887} C_VEL
LIN {X 0,Y 320.524,Z 297.81,A -85,B 0,C 180,E1 -15327.241,E2 -15327.241} C_VEL
LIN {X 0,Y 322.688,Z 300.036,A -85,B 0,C 180,E1 -15327.873,E2 -15327.873} C_VEL
LIN {X 0,Y 323.577,Z 300.84,A -85,B 0,C 180,E1 -15328.123,E2 -15328.123} C_VEL
LIN {X 0,Y 325.641,Z 304.087,A -85,B 0,C 180,E1 -15328.743,E2 -15328.743} C_VEL
LIN {X 0,Y 327.437,Z 305.894,A -85,B 0,C 180,E1 -15329.23,E2 -15329.23} C_VEL
LIN {X 0,Y 330.001,Z 309.466,A -85,B 0,C 180,E1 -15329.939,E2 -15329.939} C_VEL
LIN {X 0,Y 331.625,Z 311.561,A -85,B 0,C 180,E1 -15330.371,E2 -15330.371} C_VEL
LIN {X 0,Y 338.304,Z 320.553,A -85,B 0,C 180,E1 -15332.077,E2 -15332.077} C_VEL
LIN {X 0,Y 346.403,Z 332.266,A -85,B 0,C 180,E1 -15334.001,E2 -15334.001} C_VEL
LIN {X 0,Y 351.174,Z 339.993,A -85,B 0,C 180,E1 -15335.083,E2 -15335.083} C_VEL
LIN {X 0,Y 359.024,Z 354.201,A -85,B 0,C 180,E1 -15336.791,E2 -15336.791} C_VEL
LIN {X 0,Y 360.479,Z 357.01,A -85,B 0,C 180,E1 -15337.098,E2 -15337.098} C_VEL
LIN {X 0,Y 354.256,Z 496.634,A -85,B 0,C 180,E1 -15340.007,E2 -15340.007} C_VEL
LIN {X 0,Y 352.956,Z 511.632,A -85,B 0,C 180,E1 -15340.502,E2 -15340.502} C_VEL
LIN {X 0,Y 350.99,Z 527.881,A -85,B 0,C 180,E1 -15341.237,E2 -15341.237} C_VEL
LIN {X 0,Y 348.608,Z 543.706,A -85,B 0,C 180,E1 -15342.193,E2 -15342.193} C_VEL
LIN {X 0,Y 345.927,Z 558.685,A -85,B 0,C 180,E1 -15343.341,E2 -15343.341} C_VEL
LIN {X 0,Y 342.74,Z 573.664,A -85,B 0,C 180,E1 -15344.765,E2 -15344.765} C_VEL
LIN {X 0,Y 339.444,Z 587.552,A -85,B 0,C 180,E1 -15346.381,E2 -15346.381} C_VEL
LIN {X 0,Y 336.078,Z 600.525,A -85,B 0,C 180,E1 -15348.198,E2 -15348.198} C_VEL
LIN {X 0,Y 333.145,Z 611.166,A -85,B 0,C 180,E1 -15349.952,E2 -15349.952} C_VEL
LIN {X 0,Y 329.903,Z 622.268,A -85,B 0,C 180,E1 -15352.138,E2 -15352.138} C_VEL
LIN {X 0,Y 326.913,Z 632.332,A -85,B 0,C 180,E1 -15354.518,E2 -15354.518} C_VEL
LIN {X 0,Y 324.248,Z 641.638,A -85,B 0,C 180,E1 -15357.189,E2 -15357.189} C_VEL
LIN {X 0,Y 322.069,Z 649.305,A -85,B 0,C 180,E1 -15359.875,E2 -15359.875} C_VEL
LIN {X 0,Y 320.449,Z 655.555,A -85,B 0,C 180,E1 -15362.576,E2 -15362.576} C_VEL
LIN {X 0,Y 319.215,Z 660.418,A -85,B 0,C 180,E1 -15365.272,E2 -15365.272} C_VEL
LIN {X 0,Y 318.443,Z 664.135,A -85,B 0,C 180,E1 -15367.964,E2 -15367.964} C_VEL
LIN {X 0,Y 317.91,Z 666.734,A -85,B 0,C 180,E1 -15370.634,E2 -15370.634} C_VEL
LIN {X 0,Y 317.668,Z 668.239,A -85,B 0,C 180,E1 -15373.285,E2 -15373.285} C_VEL
LIN {X 0,Y 317.611,Z 668.787,A -85,B 0,C 180,E1 -15375.912,E2 -15375.912} C_VEL
LIN {X 0,Y 317.646,Z 668.258,A -85,B 0,C 180,E1 -15378.514,E2 -15378.514} C_VEL
LIN {X 0,Y 317.675,Z 666.844,A -85,B 0,C 180,E1 -15381.091,E2 -15381.091} C_VEL
LIN {X 0,Y 318.05,Z 664.034,A -85,B 0,C 180,E1 -15383.926,E2 -15383.926} C_VEL
LIN {X 0,Y 318.43,Z 659.864,A -85,B 0,C 180,E1 -15386.837,E2 -15386.837} C_VEL
LIN {X 0,Y 319.018,Z 655.135,A -85,B 0,C 180,E1 -15389.369,E2 -15389.369} C_VEL
LIN {X 0,Y 320.054,Z 649.179,A -85,B 0,C 180,E1 -15391.887,E2 -15391.887} C_VEL
LIN {X 0,Y 321.298,Z 642.02,A -85,B 0,C 180,E1 -15394.391,E2 -15394.391} C_VEL
LIN {X 0,Y 323.166,Z 633.464,A -85,B 0,C 180,E1 -15396.869,E2 -15396.869} C_VEL
LIN {X 0,Y 325.434,Z 623.26,A -85,B 0,C 180,E1 -15399.321,E2 -15399.321} C_VEL
LIN {X 0,Y 327.649,Z 612.705,A -85,B 0,C 180,E1 -15401.444,E2 -15401.444} C_VEL
LIN {X 0,Y 330.21,Z 600.355,A -85,B 0,C 180,E1 -15403.539,E2 -15403.539} C_VEL
LIN {X 0,Y 332.708,Z 587.932,A -85,B 0,C 180,E1 -15405.31,E2 -15405.31} C_VEL
LIN {X 0,Y 334.935,Z 575.838,A -85,B 0,C 180,E1 -15406.769,E2 -15406.769} C_VEL
LIN {X 0,Y 337.421,Z 561.487,A -85,B 0,C 180,E1 -15408.206,E2 -15408.206} C_VEL
LIN {X 0,Y 339.671,Z 545.875,A -85,B 0,C 180,E1 -15409.489,E2 -15409.489} C_VEL
LIN {X 0,Y 341.582,Z 530.8,A -85,B 0,C 180,E1 -15410.473,E2 -15410.473} C_VEL
LIN {X 0,Y 343.287,Z 514.049,A -85,B 0,C 180,E1 -15411.308,E2 -15411.308} C_VEL
LIN {X 0,Y 344.604,Z 497.157,A -85,B 0,C 180,E1 -15411.89,E2 -15411.89} C_VEL
LIN {X 0,Y 345.953,Z 461.581,A -85,B 0,C 180,E1 -15412.665,E2 -15412.665} C_VEL
LIN {X 0,Y 346.301,Z 452.063,A -85,B 0,C 180,E1 -15412.86,E2 -15412.86} C_VEL
LIN {X 0,Y 345.974,Z 446.265,A -85,B 0,C 180,E1 -15413.034,E2 -15413.034} C_VEL
LIN {X 0,Y 341.735,Z 427.663,A -85,B 0,C 180,E1 -15413.942,E2 -15413.942} C_VEL
LIN {X 0,Y 341.33,Z 421.868,A -85,B 0,C 180,E1 -15414.13,E2 -15414.13} C_VEL
LIN {X 0,Y 343.955,Z 353.02,A -85,B 0,C 180,E1 -15415.554,E2 -15415.554} C_VEL
LIN {X 0,Y 341.083,Z 346.346,A -85,B 0,C 180,E1 -15416.056,E2 -15416.056} C_VEL
LIN {X 0,Y 333.434,Z 330.933,A -85,B 0,C 180,E1 -15417.388,E2 -15417.388} C_VEL
LIN {X 0,Y 323.3,Z 313.766,A -85,B 0,C 180,E1 -15419.186,E2 -15419.186} C_VEL
LIN {X 0,Y 316.626,Z 303.364,A -85,B 0,C 180,E1 -15420.433,E2 -15420.433} C_VEL
LIN {X 0,Y 314.559,Z 300.027,A -85,B 0,C 180,E1 -15420.837,E2 -15420.837} C_VEL
LIN {X 0,Y 312.942,Z 297.585,A -85,B 0,C 180,E1 -15421.152,E2 -15421.152} C_VEL
LIN {X 0,Y 312.502,Z 295.87,A -85,B 0,C 180,E1 -15421.283,E2 -15421.283} C_VEL
LIN {X 0,Y 312.508,Z 295.865,A -85,B 0,C 180,E1 -15424.21,E2 -15424.21} C_VEL
LIN {X 0,Y 312.512,Z 295.865,A -85,B 0,C 180,E1 -15427.387,E2 -15427.387} C_VEL
LIN {X 0,Y 312.442,Z 295.876,A -85,B 0,C 180,E1 -15430.717,E2 -15430.717} C_VEL
LIN {X 0,Y 312.452,Z 295.878,A -85,B 0,C 180,E1 -15434.209,E2 -15434.209} C_VEL
LIN {X 0,Y 312.455,Z 295.871,A -85,B 0,C 180,E1 -15437.924,E2 -15437.924} C_VEL
LIN {X 0,Y 312.477,Z 295.829,A -85,B 0,C 180,E1 -15441.924,E2 -15441.924} C_VEL
LIN {X 0,Y 312.531,Z 295.814,A -85,B 0,C 180,E1 -15444.219,E2 -15444.219} C_VEL
LIN {X 0,Y 312.503,Z 295.866,A -85,B 0,C 180,E1 -15447.333,E2 -15447.333} C_VEL
LIN {X 0,Y 312.486,Z 295.856,A -85,B 0,C 180,E1 -15451.298,E2 -15451.298} C_VEL
LIN {X 0,Y 312.547,Z 295.861,A -85,B 0,C 180,E1 -15454.707,E2 -15454.707} C_VEL
LIN {X 0,Y 312.528,Z 295.866,A -85,B 0,C 180,E1 -15458.911,E2 -15458.911} C_VEL
LIN {X 0,Y 312.583,Z 295.844,A -85,B 0,C 180,E1 -15461.652,E2 -15461.652} C_VEL
LIN {X 0,Y 312.687,Z 295.847,A -85,B 0,C 180,E1 -15465.685,E2 -15465.685} C_VEL
LIN {X 0,Y 312.699,Z 295.837,A -85,B 0,C 180,E1 -15469.641,E2 -15469.641} C_VEL
LIN {X 0,Y 312.879,Z 295.806,A -85,B 0,C 180,E1 -15473.551,E2 -15473.551} C_VEL
LIN {X 0,Y 312.924,Z 295.821,A -85,B 0,C 180,E1 -15477.425,E2 -15477.425} C_VEL
LIN {X 0,Y 313.083,Z 295.778,A -85,B 0,C 180,E1 -15479.999,E2 -15479.999} C_VEL
LIN {X 0,Y 312.936,Z 295.814,A -85,B 0,C 180,E1 -15482.574,E2 -15482.574} C_VEL
LIN {X 0,Y 312.884,Z 295.797,A -85,B 0,C 180,E1 -15486.448,E2 -15486.448} C_VEL
LIN {X 0,Y 312.767,Z 295.827,A -85,B 0,C 180,E1 -15489.049,E2 -15489.049} C_VEL
LIN {X 0,Y 312.634,Z 295.85,A -85,B 0,C 180,E1 -15492.99,E2 -15492.99} C_VEL
LIN {X 0,Y 312.621,Z 295.852,A -85,B 0,C 180,E1 -15495.65,E2 -15495.65} C_VEL
LIN {X 0,Y 312.578,Z 295.861,A -85,B 0,C 180,E1 -15499.709,E2 -15499.709} C_VEL
LIN {X 0,Y 312.545,Z 295.863,A -85,B 0,C 180,E1 -15502.789,E2 -15502.789} C_VEL
LIN {X 0,Y 312.601,Z 295.86,A -85,B 0,C 180,E1 -15505.935,E2 -15505.935} C_VEL
LIN {X 0,Y 312.537,Z 295.868,A -85,B 0,C 180,E1 -15509.65,E2 -15509.65} C_VEL
LIN {X 0,Y 312.518,Z 295.868,A -85,B 0,C 180,E1 -15513.688,E2 -15513.688} C_VEL
LIN {X 0,Y 312.524,Z 295.855,A -85,B 0,C 180,E1 -15517.385,E2 -15517.385} C_VEL
LIN {X 0,Y 312.488,Z 295.861,A -85,B 0,C 180,E1 -15520.709,E2 -15520.709} C_VEL
LIN {X 0,Y 312.509,Z 296.038,A -85,B 0,C 180,E1 -15524.029,E2 -15524.029} C_VEL
LIN {X 0,Y 315.649,Z 304.556,A -85,B 0,C 180,E1 -15526.074,E2 -15526.074} C_VEL
LIN {X 0,Y 325.909,Z 322.783,A -85,B 0,C 180,E1 -15528.031,E2 -15528.031} C_VEL
LIN {X 0,Y 335.989,Z 342.978,A -85,B 0,C 180,E1 -15529.861,E2 -15529.861} C_VEL
LIN {X 0,Y 343.735,Z 360.11,A -85,B 0,C 180,E1 -15531.214,E2 -15531.214} C_VEL
LIN {X 0,Y 342.354,Z 402.17,A -85,B 0,C 180,E1 -15532.109,E2 -15532.109} C_VEL
LIN {X 0,Y 338.336,Z 512.101,A -85,B 0,C 180,E1 -15534.435,E2 -15534.435} C_VEL
LIN {X 0,Y 336.972,Z 529.111,A -85,B 0,C 180,E1 -15535.002,E2 -15535.002} C_VEL
LIN {X 0,Y 335.301,Z 544.303,A -85,B 0,C 180,E1 -15535.715,E2 -15535.715} C_VEL
LIN {X 0,Y 333.318,Z 559.706,A -85,B 0,C 180,E1 -15536.666,E2 -15536.666} C_VEL
LIN {X 0,Y 330.998,Z 573.955,A -85,B 0,C 180,E1 -15537.76,E2 -15537.76} C_VEL
LIN {X 0,Y 328.548,Z 588.115,A -85,B 0,C 180,E1 -15539.111,E2 -15539.111} C_VEL
LIN {X 0,Y 325.674,Z 602.602,A -85,B 0,C 180,E1 -15540.775,E2 -15540.775} C_VEL
LIN {X 0,Y 323.166,Z 614.935,A -85,B 0,C 180,E1 -15542.475,E2 -15542.475} C_VEL
LIN {X 0,Y 320.289,Z 628.206,A -85,B 0,C 180,E1 -15544.667,E2 -15544.667} C_VEL
LIN {X 0,Y 317.829,Z 639.377,A -85,B 0,C 180,E1 -15546.89,E2 -15546.89} C_VEL
LIN {X 0,Y 315.771,Z 649.108,A -85,B 0,C 180,E1 -15549.191,E2 -15549.191} C_VEL
LIN {X 0,Y 313.988,Z 658.182,A -85,B 0,C 180,E1 -15551.738,E2 -15551.738} C_VEL
LIN {X 0,Y 312.606,Z 665.924,A -85,B 0,C 180,E1 -15554.349,E2 -15554.349} C_VEL
LIN {X 0,Y 311.666,Z 672.22,A -85,B 0,C 180,E1 -15556.968,E2 -15556.968} C_VEL
LIN {X 0,Y 311.009,Z 677.341,A -85,B 0,C 180,E1 -15559.585,E2 -15559.585} C_VEL
LIN {X 0,Y 310.772,Z 681.327,A -85,B 0,C 180,E1 -15562.202,E2 -15562.202} C_VEL
LIN {X 0,Y 310.684,Z 684.216,A -85,B 0,C 180,E1 -15564.809,E2 -15564.809} C_VEL
LIN {X 0,Y 310.676,Z 686.112,A -85,B 0,C 180,E1 -15567.407,E2 -15567.407} C_VEL
LIN {X 0,Y 310.689,Z 686.972,A -85,B 0,C 180,E1 -15570,E2 -15570} C_VEL
LIN {X 0,Y 310.668,Z 686.899,A -85,B 0,C 180,E1 -15572.593,E2 -15572.593} C_VEL
LIN {X 0,Y 310.72,Z 685.552,A -85,B 0,C 180,E1 -15575.616,E2 -15575.616} C_VEL
LIN {X 0,Y 310.777,Z 683.811,A -85,B 0,C 180,E1 -15577.798,E2 -15577.798} C_VEL
LIN {X 0,Y 311.076,Z 680.779,A -85,B 0,C 180,E1 -15580.413,E2 -15580.413} C_VEL
LIN {X 0,Y 311.822,Z 676.766,A -85,B 0,C 180,E1 -15583.026,E2 -15583.026} C_VEL
LIN {X 0,Y 312.856,Z 671.613,A -85,B 0,C 180,E1 -15585.639,E2 -15585.639} C_VEL
LIN {X 0,Y 314.446,Z 665.38,A -85,B 0,C 180,E1 -15588.235,E2 -15588.235} C_VEL
LIN {X 0,Y 316.503,Z 657.79,A -85,B 0,C 180,E1 -15590.811,E2 -15590.811} C_VEL
LIN {X 0,Y 319.133,Z 648.773,A -85,B 0,C 180,E1 -15593.353,E2 -15593.353} C_VEL
LIN {X 0,Y 322.302,Z 638.093,A -85,B 0,C 180,E1 -15595.856,E2 -15595.856} C_VEL
LIN {X 0,Y 325.565,Z 627.076,A -85,B 0,C 180,E1 -15598.014,E2 -15598.014} C_VEL
LIN {X 0,Y 329.21,Z 614.201,A -85,B 0,C 180,E1 -15600.111,E2 -15600.111} C_VEL
LIN {X 0,Y 332.87,Z 601.067,A -85,B 0,C 180,E1 -15601.859,E2 -15601.859} C_VEL
LIN {X 0,Y 335.937,Z 588.551,A -85,B 0,C 180,E1 -15603.274,E2 -15603.274} C_VEL
LIN {X 0,Y 339.131,Z 574.763,A -85,B 0,C 180,E1 -15604.563,E2 -15604.563} C_VEL
LIN {X 0,Y 341.978,Z 560.185,A -85,B 0,C 180,E1 -15605.672,E2 -15605.672} C_VEL
LIN {X 0,Y 344.598,Z 544.405,A -85,B 0,C 180,E1 -15606.623,E2 -15606.623} C_VEL
LIN {X 0,Y 346.857,Z 528.245,A -85,B 0,C 180,E1 -15607.344,E2 -15607.344} C_VEL
LIN {X 0,Y 348.381,Z 512.992,A -85,B 0,C 180,E1 -15607.839,E2 -15607.839} C_VEL
LIN {X 0,Y 350.864,Z 459.991,A -85,B 0,C 180,E1 -15608.983,E2 -15608.983} C_VEL
LIN {X 0,Y 355.056,Z 367.044,A -85,B 0,C 180,E1 -15610.932,E2 -15610.932} C_VEL
LIN {X 0,Y 347.514,Z 352.246,A -85,B 0,C 180,E1 -15612.64,E2 -15612.64} C_VEL
LIN {X 0,Y 340.131,Z 339.178,A -85,B 0,C 180,E1 -15614.407,E2 -15614.407} C_VEL
LIN {X 0,Y 332.726,Z 327.32,A -85,B 0,C 180,E1 -15616.299,E2 -15616.299} C_VEL
LIN {X 0,Y 327.049,Z 318.873,A -85,B 0,C 180,E1 -15617.841,E2 -15617.841} C_VEL
LIN {X 0,Y 319.331,Z 307.895,A -85,B 0,C 180,E1 -15620.12,E2 -15620.12} C_VEL
LIN {X 0,Y 315.104,Z 302.138,A -85,B 0,C 180,E1 -15621.539,E2 -15621.539} C_VEL
LIN {X 0,Y 312.515,Z 295.859,A -85,B 0,C 180,E1 -15623.972,E2 -15623.972} C_VEL
LIN {X 0,Y 312.503,Z 295.846,A -85,B 0,C 180,E1 -15627.334,E2 -15627.334} C_VEL
LIN {X 0,Y 312.544,Z 295.838,A -85,B 0,C 180,E1 -15631.28,E2 -15631.28} C_VEL
LIN {X 0,Y 312.585,Z 295.861,A -85,B 0,C 180,E1 -15634.712,E2 -15634.712} C_VEL
LIN {X 0,Y 312.539,Z 295.848,A -85,B 0,C 180,E1 -15638.913,E2 -15638.913} C_VEL
LIN {X 0,Y 312.639,Z 295.833,A -85,B 0,C 180,E1 -15641.657,E2 -15641.657} C_VEL
LIN {X 0,Y 312.695,Z 295.845,A -85,B 0,C 180,E1 -15645.687,E2 -15645.687} C_VEL
